LIN {X 0,Y 474.681,Z 256.169,A -85,B 0,C 180,E1 -7215.456,E2 -7215.456} C_VEL
LIN {X 0,Y 474.597,Z 256.179,A -85,B 0,C 180,E1 -7219.013,E2 -7219.013} C_VEL
LIN {X 0,Y 474.568,Z 256.186,A -85,B 0,C 180,E1 -7221.73,E2 -7221.73} C_VEL
LIN {X 0,Y 474.615,Z 256.175,A -85,B 0,C 180,E1 -7224.495,E2 -7224.495} C_VEL
LIN {X 0,Y 474.59,Z 256.182,A -85,B 0,C 180,E1 -7227.327,E2 -7227.327} C_VEL
LIN {X 0,Y 474.543,Z 256.184,A -85,B 0,C 180,E1 -7230.234,E2 -7230.234} C_VEL
LIN {X 0,Y 474.608,Z 256.18,A -85,B 0,C 180,E1 -7233.223,E2 -7233.223} C_VEL
LIN {X 0,Y 474.566,Z 256.181,A -85,B 0,C 180,E1 -7236.325,E2 -7236.325} C_VEL
LIN {X 0,Y 474.594,Z 256.179,A -85,B 0,C 180,E1 -7239.644,E2 -7239.644} C_VEL
LIN {X 0,Y 474.564,Z 256.185,A -85,B 0,C 180,E1 -7242.94,E2 -7242.94} C_VEL
LIN {X 0,Y 474.575,Z 256.179,A -85,B 0,C 180,E1 -7245.892,E2 -7245.892} C_VEL
LIN {X 0,Y 474.594,Z 256.183,A -85,B 0,C 180,E1 -7249.045,E2 -7249.045} C_VEL
LIN {X 0,Y 474.585,Z 256.178,A -85,B 0,C 180,E1 -7251.708,E2 -7251.708} C_VEL
LIN {X 0,Y 474.604,Z 256.181,A -85,B 0,C 180,E1 -7254.725,E2 -7254.725} C_VEL
LIN {X 0,Y 474.605,Z 256.175,A -85,B 0,C 180,E1 -7257.786,E2 -7257.786} C_VEL
LIN {X 0,Y 474.571,Z 256.185,A -85,B 0,C 180,E1 -7260.896,E2 -7260.896} C_VEL
LIN {X 0,Y 474.567,Z 256.182,A -85,B 0,C 180,E1 -7263.623,E2 -7263.623} C_VEL
LIN {X 0,Y 474.649,Z 256.338,A -85,B 0,C 180,E1 -7265.391,E2 -7265.391} C_VEL
LIN {X 0,Y 475.967,Z 264.349,A -85,B 0,C 180,E1 -7266.966,E2 -7266.966} C_VEL
LIN {X 0,Y 475.506,Z 278.927,A -85,B 0,C 180,E1 -7269.676,E2 -7269.676} C_VEL
LIN {X 0,Y 475.135,Z 292.245,A -85,B 0,C 180,E1 -7272.127,E2 -7272.127} C_VEL
LIN {X 0,Y 474.672,Z 310.333,A -85,B 0,C 180,E1 -7275.422,E2 -7275.422} C_VEL
LIN {X 0,Y 474.437,Z 318.145,A -85,B 0,C 180,E1 -7276.819,E2 -7276.819} C_VEL
LIN {X 0,Y 476.321,Z 335.84,A -85,B 0,C 180,E1 -7277.139,E2 -7277.139} C_VEL
LIN {X 0,Y 475.981,Z 395.396,A -85,B 0,C 180,E1 -7278.051,E2 -7278.051} C_VEL
LIN {X 0,Y 475.775,Z 405.125,A -85,B 0,C 180,E1 -7278.309,E2 -7278.309} C_VEL
LIN {X 0,Y 475.51,Z 415.201,A -85,B 0,C 180,E1 -7278.707,E2 -7278.707} C_VEL
LIN {X 0,Y 475.139,Z 426.652,A -85,B 0,C 180,E1 -7279.346,E2 -7279.346} C_VEL
LIN {X 0,Y 474.877,Z 435.271,A -85,B 0,C 180,E1 -7279.986,E2 -7279.986} C_VEL
LIN {X 0,Y 474.58,Z 443.381,A -85,B 0,C 180,E1 -7280.733,E2 -7280.733} C_VEL
LIN {X 0,Y 474.351,Z 450.086,A -85,B 0,C 180,E1 -7281.48,E2 -7281.48} C_VEL
LIN {X 0,Y 474.147,Z 456.454,A -85,B 0,C 180,E1 -7282.334,E2 -7282.334} C_VEL
LIN {X 0,Y 474.037,Z 461.751,A -85,B 0,C 180,E1 -7283.189,E2 -7283.189} C_VEL
LIN {X 0,Y 473.901,Z 466.167,A -85,B 0,C 180,E1 -7284.042,E2 -7284.042} C_VEL
LIN {X 0,Y 473.795,Z 471.377,A -85,B 0,C 180,E1 -7285.321,E2 -7285.321} C_VEL
LIN {X 0,Y 473.848,Z 475.21,A -85,B 0,C 180,E1 -7286.599,E2 -7286.599} C_VEL
LIN {X 0,Y 473.786,Z 476.969,A -85,B 0,C 180,E1 -7287.45,E2 -7287.45} C_VEL
LIN {X 0,Y 473.757,Z 478.23,A -85,B 0,C 180,E1 -7288.3,E2 -7288.3} C_VEL
LIN {X 0,Y 473.695,Z 479.012,A -85,B 0,C 180,E1 -7289.15,E2 -7289.15} C_VEL
LIN {X 0,Y 473.684,Z 479.309,A -85,B 0,C 180,E1 -7290,E2 -7290} C_VEL
LIN {X 0,Y 473.695,Z 479.011,A -85,B 0,C 180,E1 -7290.851,E2 -7290.851} C_VEL
LIN {X 0,Y 473.757,Z 478.227,A -85,B 0,C 180,E1 -7291.701,E2 -7291.701} C_VEL
LIN {X 0,Y 473.787,Z 476.965,A -85,B 0,C 180,E1 -7292.551,E2 -7292.551} C_VEL
LIN {X 0,Y 473.842,Z 474.041,A -85,B 0,C 180,E1 -7293.827,E2 -7293.827} C_VEL
LIN {X 0,Y 473.795,Z 471.371,A -85,B 0,C 180,E1 -7294.68,E2 -7294.68} C_VEL
LIN {X 0,Y 473.9,Z 466.157,A -85,B 0,C 180,E1 -7295.959,E2 -7295.959} C_VEL
LIN {X 0,Y 474.108,Z 459.292,A -85,B 0,C 180,E1 -7297.239,E2 -7297.239} C_VEL
LIN {X 0,Y 474.301,Z 451.789,A -85,B 0,C 180,E1 -7298.307,E2 -7298.307} C_VEL
LIN {X 0,Y 474.532,Z 444.396,A -85,B 0,C 180,E1 -7299.162,E2 -7299.162} C_VEL
LIN {X 0,Y 474.818,Z 436.486,A -85,B 0,C 180,E1 -7299.908,E2 -7299.908} C_VEL
LIN {X 0,Y 475.064,Z 428.131,A -85,B 0,C 180,E1 -7300.549,E2 -7300.549} C_VEL
LIN {X 0,Y 475.485,Z 417.478,A -85,B 0,C 180,E1 -7301.187,E2 -7301.187} C_VEL
LIN {X 0,Y 475.719,Z 406.729,A -85,B 0,C 180,E1 -7301.64,E2 -7301.64} C_VEL
LIN {X 0,Y 475.995,Z 396.227,A -85,B 0,C 180,E1 -7301.93,E2 -7301.93} C_VEL
LIN {X 0,Y 476.23,Z 334.22,A -85,B 0,C 180,E1 -7302.887,E2 -7302.887} C_VEL
LIN {X 0,Y 474.453,Z 318.027,A -85,B 0,C 180,E1 -7303.184,E2 -7303.184} C_VEL
LIN {X 0,Y 474.813,Z 302.683,A -85,B 0,C 180,E1 -7305.967,E2 -7305.967} C_VEL
LIN {X 0,Y 475.369,Z 286.185,A -85,B 0,C 180,E1 -7308.981,E2 -7308.981} C_VEL
LIN {X 0,Y 475.865,Z 269.199,A -85,B 0,C 180,E1 -7312.124,E2 -7312.124} C_VEL
LIN {X 0,Y 475.822,Z 263.099,A -85,B 0,C 180,E1 -7313.273,E2 -7313.273} C_VEL
LIN {X 0,Y 474.632,Z 256.175,A -85,B 0,C 180,E1 -7314.67,E2 -7314.67} C_VEL
LIN {X 0,Y 474.588,Z 256.177,A -85,B 0,C 180,E1 -7318.287,E2 -7318.287} C_VEL
LIN {X 0,Y 474.573,Z 256.186,A -85,B 0,C 180,E1 -7321.22,E2 -7321.22} C_VEL
LIN {X 0,Y 474.604,Z 256.175,A -85,B 0,C 180,E1 -7324.244,E2 -7324.244} C_VEL
LIN {X 0,Y 474.533,Z 256.188,A -85,B 0,C 180,E1 -7327.389,E2 -7327.389} C_VEL
LIN {X 0,Y 474.578,Z 256.18,A -85,B 0,C 180,E1 -7329.64,E2 -7329.64} C_VEL
LIN {X 0,Y 474.565,Z 256.187,A -85,B 0,C 180,E1 -7332.94,E2 -7332.94} C_VEL
LIN {X 0,Y 474.58,Z 256.179,A -85,B 0,C 180,E1 -7335.892,E2 -7335.892} C_VEL
LIN {X 0,Y 474.586,Z 256.182,A -85,B 0,C 180,E1 -7339.047,E2 -7339.047} C_VEL
LIN {X 0,Y 474.586,Z 256.178,A -85,B 0,C 180,E1 -7341.708,E2 -7341.708} C_VEL
LIN {X 0,Y 474.607,Z 256.182,A -85,B 0,C 180,E1 -7344.724,E2 -7344.724} C_VEL
LIN {X 0,Y 474.609,Z 256.175,A -85,B 0,C 180,E1 -7347.786,E2 -7347.786} C_VEL
LIN {X 0,Y 474.575,Z 256.183,A -85,B 0,C 180,E1 -7350.896,E2 -7350.896} C_VEL
LIN {X 0,Y 474.571,Z 256.18,A -85,B 0,C 180,E1 -7353.623,E2 -7353.623} C_VEL
LIN {X 0,Y 474.596,Z 256.181,A -85,B 0,C 180,E1 -7356.653,E2 -7356.653} C_VEL
LIN {X 0,Y 474.586,Z 256.181,A -85,B 0,C 180,E1 -7360.087,E2 -7360.087} C_VEL
LIN {X 0,Y 474.582,Z 256.181,A -85,B 0,C 180,E1 -7362.772,E2 -7362.772} C_VEL
LIN {X 0,Y 474.601,Z 256.177,A -85,B 0,C 180,E1 -7365.42,E2 -7365.42} C_VEL
LIN {X 0,Y 474.685,Z 256.171,A -85,B 0,C 180,E1 -7368.037,E2 -7368.037} C_VEL
LIN {X 0,Y 474.661,Z 256.17,A -85,B 0,C 180,E1 -7371.485,E2 -7371.485} C_VEL
LIN {X 0,Y 474.735,Z 256.165,A -85,B 0,C 180,E1 -7374.052,E2 -7374.052} C_VEL
LIN {X 0,Y 474.871,Z 256.144,A -85,B 0,C 180,E1 -7377.455,E2 -7377.455} C_VEL
LIN {X 0,Y 474.88,Z 256.146,A -85,B 0,C 180,E1 -7380,E2 -7380} C_VEL
LIN {X 0,Y 474.871,Z 256.146,A -85,B 0,C 180,E1 -7382.545,E2 -7382.545} C_VEL
LIN {X 0,Y 474.736,Z 256.163,A -85,B 0,C 180,E1 -7385.948,E2 -7385.948} C_VEL
LIN {X 0,Y 474.662,Z 256.172,A -85,B 0,C 180,E1 -7388.515,E2 -7388.515} C_VEL
LIN {X 0,Y 474.694,Z 256.168,A -85,B 0,C 180,E1 -7391.963,E2 -7391.963} C_VEL
LIN {X 0,Y 474.689,Z 256.17,A -85,B 0,C 180,E1 -7395.456,E2 -7395.456} C_VEL
LIN {X 0,Y 474.604,Z 256.178,A -85,B 0,C 180,E1 -7399.013,E2 -7399.013} C_VEL
LIN {X 0,Y 474.576,Z 256.183,A -85,B 0,C 180,E1 -7401.73,E2 -7401.73} C_VEL
LIN {X 0,Y 474.626,Z 256.175,A -85,B 0,C 180,E1 -7404.495,E2 -7404.495} C_VEL
LIN {X 0,Y 474.598,Z 256.181,A -85,B 0,C 180,E1 -7407.326,E2 -7407.326} C_VEL
LIN {X 0,Y 474.585,Z 256.18,A -85,B 0,C 180,E1 -7410.232,E2 -7410.232} C_VEL
LIN {X 0,Y 474.616,Z 256.178,A -85,B 0,C 180,E1 -7413.222,E2 -7413.222} C_VEL
LIN {X 0,Y 474.583,Z 256.18,A -85,B 0,C 180,E1 -7416.324,E2 -7416.324} C_VEL
LIN {X 0,Y 474.602,Z 256.181,A -85,B 0,C 180,E1 -7419.643,E2 -7419.643} C_VEL
LIN {X 0,Y 474.57,Z 256.184,A -85,B 0,C 180,E1 -7422.939,E2 -7422.939} C_VEL
LIN {X 0,Y 474.603,Z 256.178,A -85,B 0,C 180,E1 -7425.894,E2 -7425.894} C_VEL
LIN {X 0,Y 474.592,Z 256.182,A -85,B 0,C 180,E1 -7429.339,E2 -7429.339} C_VEL
LIN {X 0,Y 474.607,Z 256.178,A -85,B 0,C 180,E1 -7431.705,E2 -7431.705} C_VEL
LIN {X 0,Y 474.621,Z 256.177,A -85,B 0,C 180,E1 -7434.725,E2 -7434.725} C_VEL
LIN {X 0,Y 474.623,Z 256.175,A -85,B 0,C 180,E1 -7437.786,E2 -7437.786} C_VEL
LIN {X 0,Y 474.595,Z 256.181,A -85,B 0,C 180,E1 -7440.891,E2 -7440.891} C_VEL
LIN {X 0,Y 474.591,Z 256.179,A -85,B 0,C 180,E1 -7443.624,E2 -7443.624} C_VEL
LIN {X 0,Y 474.635,Z 256.175,A -85,B 0,C 180,E1 -7446.642,E2 -7446.642} C_VEL
LIN {X 0,Y 474.65,Z 256.173,A -85,B 0,C 180,E1 -7450.089,E2 -7450.089} C_VEL
LIN {X 0,Y 474.642,Z 256.172,A -85,B 0,C 180,E1 -7451.629,E2 -7451.629} C_VEL
LIN {X 0,Y 473.94,Z 256.262,A -85,B 0,C 180,E1 -7452.101,E2 -7452.101} C_VEL
LIN {X 0,Y 471.046,Z 256.625,A -85,B 0,C 180,E1 -7452.839,E2 -7452.839} C_VEL
LIN {X 0,Y 468.163,Z 256.982,A -85,B 0,C 180,E1 -7453.585,E2 -7453.585} C_VEL
LIN {X 0,Y 467.499,Z 257.066,A -85,B 0,C 180,E1 -7454.067,E2 -7454.067} C_VEL
LIN {X 0,Y 467.577,Z 257.787,A -85,B 0,C 180,E1 -7454.302,E2 -7454.302} C_VEL
LIN {X 0,Y 467.519,Z 268.24,A -85,B 0,C 180,E1 -7456.658,E2 -7456.658} C_VEL
LIN {X 0,Y 469.716,Z 281.044,A -85,B 0,C 180,E1 -7456.941,E2 -7456.941} C_VEL
LIN {X 0,Y 469.21,Z 344.335,A -85,B 0,C 180,E1 -7457.922,E2 -7457.922} C_VEL
LIN {X 0,Y 469.077,Z 353.451,A -85,B 0,C 180,E1 -7458.166,E2 -7458.166} C_VEL
LIN {X 0,Y 468.936,Z 363.039,A -85,B 0,C 180,E1 -7458.546,E2 -7458.546} C_VEL
LIN {X 0,Y 468.714,Z 373.066,A -85,B 0,C 180,E1 -7459.088,E2 -7459.088} C_VEL
LIN {X 0,Y 468.48,Z 383.462,A -85,B 0,C 180,E1 -7459.847,E2 -7459.847} C_VEL
LIN {X 0,Y 468.128,Z 391.587,A -85,B 0,C 180,E1 -7460.603,E2 -7460.603} C_VEL
LIN {X 0,Y 467.835,Z 398.286,A -85,B 0,C 180,E1 -7461.36,E2 -7461.36} C_VEL
LIN {X 0,Y 467.558,Z 404.624,A -85,B 0,C 180,E1 -7462.225,E2 -7462.225} C_VEL
LIN {X 0,Y 467.426,Z 409.885,A -85,B 0,C 180,E1 -7463.091,E2 -7463.091} C_VEL
LIN {X 0,Y 467.161,Z 414.285,A -85,B 0,C 180,E1 -7463.955,E2 -7463.955} C_VEL
LIN {X 0,Y 467.088,Z 419.44,A -85,B 0,C 180,E1 -7465.253,E2 -7465.253} C_VEL
LIN {X 0,Y 466.948,Z 422.096,A -85,B 0,C 180,E1 -7466.116,E2 -7466.116} C_VEL
LIN {X 0,Y 466.845,Z 424.999,A -85,B 0,C 180,E1 -7467.411,E2 -7467.411} C_VEL
LIN {X 0,Y 466.704,Z 426.276,A -85,B 0,C 180,E1 -7468.274,E2 -7468.274} C_VEL
LIN {X 0,Y 466.636,Z 427.083,A -85,B 0,C 180,E1 -7469.137,E2 -7469.137} C_VEL
LIN {X 0,Y 466.621,Z 427.39,A -85,B 0,C 180,E1 -7470,E2 -7470} C_VEL
LIN {X 0,Y 466.636,Z 427.117,A -85,B 0,C 180,E1 -7470.863,E2 -7470.863} C_VEL
LIN {X 0,Y 466.705,Z 426.378,A -85,B 0,C 180,E1 -7471.725,E2 -7471.725} C_VEL
LIN {X 0,Y 466.844,Z 425.171,A -85,B 0,C 180,E1 -7472.588,E2 -7472.588} C_VEL
LIN {X 0,Y 466.945,Z 422.341,A -85,B 0,C 180,E1 -7473.883,E2 -7473.883} C_VEL
LIN {X 0,Y 467.069,Z 419.763,A -85,B 0,C 180,E1 -7474.747,E2 -7474.747} C_VEL
LIN {X 0,Y 467.154,Z 414.693,A -85,B 0,C 180,E1 -7476.045,E2 -7476.045} C_VEL
LIN {X 0,Y 467.456,Z 409.234,A -85,B 0,C 180,E1 -7477.123,E2 -7477.123} C_VEL
LIN {X 0,Y 467.696,Z 402.363,A -85,B 0,C 180,E1 -7478.207,E2 -7478.207} C_VEL
LIN {X 0,Y 467.994,Z 394.477,A -85,B 0,C 180,E1 -7479.181,E2 -7479.181} C_VEL
LIN {X 0,Y 468.331,Z 386.948,A -85,B 0,C 180,E1 -7479.937,E2 -7479.937} C_VEL
LIN {X 0,Y 468.521,Z 379.064,A -85,B 0,C 180,E1 -7480.588,E2 -7480.588} C_VEL
LIN {X 0,Y 468.804,Z 370.915,A -85,B 0,C 180,E1 -7481.128,E2 -7481.128} C_VEL
LIN {X 0,Y 469.019,Z 362.665,A -85,B 0,C 180,E1 -7481.561,E2 -7481.561} C_VEL
LIN {X 0,Y 469.096,Z 353.77,A -85,B 0,C 180,E1 -7481.915,E2 -7481.915} C_VEL
LIN {X 0,Y 469.262,Z 344.657,A -85,B 0,C 180,E1 -7482.161,E2 -7482.161} C_VEL
LIN {X 0,Y 469.554,Z 279.505,A -85,B 0,C 180,E1 -7483.179,E2 -7483.179} C_VEL
LIN {X 0,Y 467.522,Z 268.288,A -85,B 0,C 180,E1 -7483.427,E2 -7483.427} C_VEL
LIN {X 0,Y 467.464,Z 257.074,A -85,B 0,C 180,E1 -7485.977,E2 -7485.977} C_VEL
LIN {X 0,Y 467.608,Z 257.049,A -85,B 0,C 180,E1 -7488.761,E2 -7488.761} C_VEL
LIN {X 0,Y 467.57,Z 257.057,A -85,B 0,C 180,E1 -7491.264,E2 -7491.264} C_VEL
LIN {X 0,Y 467.549,Z 257.057,A -85,B 0,C 180,E1 -7493.944,E2 -7493.944} C_VEL
LIN {X 0,Y 467.533,Z 257.061,A -85,B 0,C 180,E1 -7496.805,E2 -7496.805} C_VEL
LIN {X 0,Y 467.53,Z 257.06,A -85,B 0,C 180,E1 -7499.739,E2 -7499.739} C_VEL
LIN {X 0,Y 467.57,Z 257.057,A -85,B 0,C 180,E1 -7502.759,E2 -7502.759} C_VEL
LIN {X 0,Y 467.546,Z 257.057,A -85,B 0,C 180,E1 -7505.89,E2 -7505.89} C_VEL
LIN {X 0,Y 467.549,Z 257.058,A -85,B 0,C 180,E1 -7509.147,E2 -7509.147} C_VEL
LIN {X 0,Y 467.555,Z 257.058,A -85,B 0,C 180,E1 -7511.404,E2 -7511.404} C_VEL
LIN {X 0,Y 467.561,Z 257.056,A -85,B 0,C 180,E1 -7515.052,E2 -7515.052} C_VEL
LIN {X 0,Y 467.556,Z 257.057,A -85,B 0,C 180,E1 -7518.725,E2 -7518.725} C_VEL
LIN {X 0,Y 467.55,Z 257.057,A -85,B 0,C 180,E1 -7521.954,E2 -7521.954} C_VEL
LIN {X 0,Y 467.55,Z 257.058,A -85,B 0,C 180,E1 -7525.166,E2 -7525.166} C_VEL
LIN {X 0,Y 467.552,Z 257.058,A -85,B 0,C 180,E1 -7528.257,E2 -7528.257} C_VEL
LIN {X 0,Y 467.534,Z 257.059,A -85,B 0,C 180,E1 -7531.247,E2 -7531.247} C_VEL
LIN {X 0,Y 467.572,Z 257.055,A -85,B 0,C 180,E1 -7534.401,E2 -7534.401} C_VEL
LIN {X 0,Y 467.563,Z 257.056,A -85,B 0,C 180,E1 -7536.995,E2 -7536.995} C_VEL
LIN {X 0,Y 467.605,Z 257.051,A -85,B 0,C 180,E1 -7539.776,E2 -7539.776} C_VEL
LIN {X 0,Y 467.562,Z 257.057,A -85,B 0,C 180,E1 -7542.505,E2 -7542.505} C_VEL
LIN {X 0,Y 467.585,Z 257.052,A -85,B 0,C 180,E1 -7545.196,E2 -7545.196} C_VEL
LIN {X 0,Y 467.642,Z 257.046,A -85,B 0,C 180,E1 -7547.854,E2 -7547.854} C_VEL
LIN {X 0,Y 467.627,Z 257.047,A -85,B 0,C 180,E1 -7551.356,E2 -7551.356} C_VEL
LIN {X 0,Y 467.697,Z 257.039,A -85,B 0,C 180,E1 -7553.962,E2 -7553.962} C_VEL
LIN {X 0,Y 467.806,Z 257.026,A -85,B 0,C 180,E1 -7557.417,E2 -7557.417} C_VEL
LIN {X 0,Y 467.843,Z 257.022,A -85,B 0,C 180,E1 -7560,E2 -7560} C_VEL
LIN {X 0,Y 467.806,Z 257.025,A -85,B 0,C 180,E1 -7562.583,E2 -7562.583} C_VEL
LIN {X 0,Y 467.694,Z 257.043,A -85,B 0,C 180,E1 -7566.038,E2 -7566.038} C_VEL
LIN {X 0,Y 467.626,Z 257.046,A -85,B 0,C 180,E1 -7568.644,E2 -7568.644} C_VEL
LIN {X 0,Y 467.642,Z 257.045,A -85,B 0,C 180,E1 -7572.354,E2 -7572.354} C_VEL
LIN {X 0,Y 467.594,Z 257.055,A -85,B 0,C 180,E1 -7575.863,E2 -7575.863} C_VEL
LIN {X 0,Y 467.546,Z 257.058,A -85,B 0,C 180,E1 -7579.311,E2 -7579.311} C_VEL
LIN {X 0,Y 467.514,Z 257.061,A -85,B 0,C 180,E1 -7582.075,E2 -7582.075} C_VEL
LIN {X 0,Y 467.55,Z 257.056,A -85,B 0,C 180,E1 -7584.89,E2 -7584.89} C_VEL
LIN {X 0,Y 467.533,Z 257.06,A -85,B 0,C 180,E1 -7587.775,E2 -7587.775} C_VEL
LIN {X 0,Y 467.523,Z 257.061,A -85,B 0,C 180,E1 -7591.037,E2 -7591.037} C_VEL
LIN {X 0,Y 467.56,Z 257.055,A -85,B 0,C 180,E1 -7593.79,E2 -7593.79} C_VEL
LIN {X 0,Y 467.5,Z 257.064,A -85,B 0,C 180,E1 -7596.965,E2 -7596.965} C_VEL
LIN {X 0,Y 467.555,Z 257.054,A -85,B 0,C 180,E1 -7599.951,E2 -7599.951} C_VEL
LIN {X 0,Y 467.513,Z 257.06,A -85,B 0,C 180,E1 -7602.568,E2 -7602.568} C_VEL
LIN {X 0,Y 467.559,Z 257.06,A -85,B 0,C 180,E1 -7605.053,E2 -7605.053} C_VEL
LIN {X 0,Y 467.555,Z 257.057,A -85,B 0,C 180,E1 -7608.726,E2 -7608.726} C_VEL
LIN {X 0,Y 467.535,Z 257.056,A -85,B 0,C 180,E1 -7611.953,E2 -7611.953} C_VEL
LIN {X 0,Y 467.54,Z 257.058,A -85,B 0,C 180,E1 -7615.166,E2 -7615.166} C_VEL
LIN {X 0,Y 467.538,Z 257.057,A -85,B 0,C 180,E1 -7618.257,E2 -7618.257} C_VEL
LIN {X 0,Y 467.52,Z 257.06,A -85,B 0,C 180,E1 -7621.247,E2 -7621.247} C_VEL
LIN {X 0,Y 467.558,Z 257.059,A -85,B 0,C 180,E1 -7624.406,E2 -7624.406} C_VEL
LIN {X 0,Y 467.598,Z 257.157,A -85,B 0,C 180,E1 -7625.232,E2 -7625.232} C_VEL
LIN {X 0,Y 468.96,Z 265.186,A -85,B 0,C 180,E1 -7626.838,E2 -7626.838} C_VEL
LIN {X 0,Y 468.586,Z 278.538,A -85,B 0,C 180,E1 -7629.363,E2 -7629.363} C_VEL
LIN {X 0,Y 468.1,Z 293.061,A -85,B 0,C 180,E1 -7632.075,E2 -7632.075} C_VEL
LIN {X 0,Y 467.656,Z 309.939,A -85,B 0,C 180,E1 -7635.199,E2 -7635.199} C_VEL
LIN {X 0,Y 467.41,Z 317.763,A -85,B 0,C 180,E1 -7636.617,E2 -7636.617} C_VEL
LIN {X 0,Y 469.384,Z 335.605,A -85,B 0,C 180,E1 -7636.947,E2 -7636.947} C_VEL
LIN {X 0,Y 469.034,Z 395.056,A -85,B 0,C 180,E1 -7637.873,E2 -7637.873} C_VEL
LIN {X 0,Y 468.823,Z 404.74,A -85,B 0,C 180,E1 -7638.133,E2 -7638.133} C_VEL
LIN {X 0,Y 468.544,Z 414.814,A -85,B 0,C 180,E1 -7638.537,E2 -7638.537} C_VEL
LIN {X 0,Y 468.151,Z 426.262,A -85,B 0,C 180,E1 -7639.185,E2 -7639.185} C_VEL
LIN {X 0,Y 467.854,Z 434.879,A -85,B 0,C 180,E1 -7639.834,E2 -7639.834} C_VEL
LIN {X 0,Y 467.553,Z 442.99,A -85,B 0,C 180,E1 -7640.592,E2 -7640.592} C_VEL
LIN {X 0,Y 467.291,Z 449.694,A -85,B 0,C 180,E1 -7641.35,E2 -7641.35} C_VEL
LIN {X 0,Y 467.076,Z 456.061,A -85,B 0,C 180,E1 -7642.218,E2 -7642.218} C_VEL
LIN {X 0,Y 466.991,Z 461.36,A -85,B 0,C 180,E1 -7643.086,E2 -7643.086} C_VEL
LIN {X 0,Y 466.811,Z 465.774,A -85,B 0,C 180,E1 -7643.951,E2 -7643.951} C_VEL
LIN {X 0,Y 466.721,Z 470.986,A -85,B 0,C 180,E1 -7645.25,E2 -7645.25} C_VEL
LIN {X 0,Y 466.761,Z 474.818,A -85,B 0,C 180,E1 -7646.548,E2 -7646.548} C_VEL
LIN {X 0,Y 466.705,Z 476.578,A -85,B 0,C 180,E1 -7647.411,E2 -7647.411} C_VEL
LIN {X 0,Y 466.692,Z 477.84,A -85,B 0,C 180,E1 -7648.275,E2 -7648.275} C_VEL
LIN {X 0,Y 466.625,Z 478.622,A -85,B 0,C 180,E1 -7649.137,E2 -7649.137} C_VEL
LIN {X 0,Y 466.612,Z 478.918,A -85,B 0,C 180,E1 -7650,E2 -7650} C_VEL
LIN {X 0,Y 466.625,Z 478.621,A -85,B 0,C 180,E1 -7650.863,E2 -7650.863} C_VEL
LIN {X 0,Y 466.692,Z 477.837,A -85,B 0,C 180,E1 -7651.726,E2 -7651.726} C_VEL
LIN {X 0,Y 466.705,Z 476.573,A -85,B 0,C 180,E1 -7652.59,E2 -7652.59} C_VEL
LIN {X 0,Y 466.732,Z 473.647,A -85,B 0,C 180,E1 -7653.886,E2 -7653.886} C_VEL
LIN {X 0,Y 466.721,Z 470.978,A -85,B 0,C 180,E1 -7654.751,E2 -7654.751} C_VEL
LIN {X 0,Y 466.81,Z 465.762,A -85,B 0,C 180,E1 -7656.05,E2 -7656.05} C_VEL
LIN {X 0,Y 467.041,Z 458.897,A -85,B 0,C 180,E1 -7657.349,E2 -7657.349} C_VEL
LIN {X 0,Y 467.237,Z 451.394,A -85,B 0,C 180,E1 -7658.434,E2 -7658.434} C_VEL
LIN {X 0,Y 467.505,Z 444.001,A -85,B 0,C 180,E1 -7659.3,E2 -7659.3} C_VEL
LIN {X 0,Y 467.825,Z 436.092,A -85,B 0,C 180,E1 -7660.058,E2 -7660.058} C_VEL
LIN {X 0,Y 468.085,Z 427.736,A -85,B 0,C 180,E1 -7660.708,E2 -7660.708} C_VEL
LIN {X 0,Y 468.52,Z 417.081,A -85,B 0,C 180,E1 -7661.355,E2 -7661.355} C_VEL
LIN {X 0,Y 468.77,Z 406.33,A -85,B 0,C 180,E1 -7661.815,E2 -7661.815} C_VEL
LIN {X 0,Y 469.054,Z 395.824,A -85,B 0,C 180,E1 -7662.109,E2 -7662.109} C_VEL
LIN {X 0,Y 469.386,Z 335.429,A -85,B 0,C 180,E1 -7663.054,E2 -7663.054} C_VEL
LIN {X 0,Y 467.395,Z 317.627,A -85,B 0,C 180,E1 -7663.386,E2 -7663.386} C_VEL
LIN {X 0,Y 467.72,Z 303.904,A -85,B 0,C 180,E1 -7665.915,E2 -7665.915} C_VEL
LIN {X 0,Y 468.338,Z 287.148,A -85,B 0,C 180,E1 -7669.022,E2 -7669.022} C_VEL
LIN {X 0,Y 468.895,Z 270.019,A -85,B 0,C 180,E1 -7672.239,E2 -7672.239} C_VEL
LIN {X 0,Y 468.82,Z 263.978,A -85,B 0,C 180,E1 -7673.396,E2 -7673.396} C_VEL
LIN {X 0,Y 467.584,Z 257.054,A -85,B 0,C 180,E1 -7674.829,E2 -7674.829} C_VEL
LIN {X 0,Y 467.537,Z 257.059,A -85,B 0,C 180,E1 -7677.775,E2 -7677.775} C_VEL
LIN {X 0,Y 467.527,Z 257.061,A -85,B 0,C 180,E1 -7681.037,E2 -7681.037} C_VEL
LIN {X 0,Y 467.562,Z 257.052,A -85,B 0,C 180,E1 -7684.238,E2 -7684.238} C_VEL
LIN {X 0,Y 467.51,Z 257.066,A -85,B 0,C 180,E1 -7687.18,E2 -7687.18} C_VEL
LIN {X 0,Y 467.517,Z 257.058,A -85,B 0,C 180,E1 -7690.271,E2 -7690.271} C_VEL
LIN {X 0,Y 467.516,Z 257.06,A -85,B 0,C 180,E1 -7692.569,E2 -7692.569} C_VEL
LIN {X 0,Y 467.562,Z 257.058,A -85,B 0,C 180,E1 -7695.052,E2 -7695.052} C_VEL
LIN {X 0,Y 467.554,Z 257.059,A -85,B 0,C 180,E1 -7698.727,E2 -7698.727} C_VEL
LIN {X 0,Y 467.537,Z 257.056,A -85,B 0,C 180,E1 -7701.953,E2 -7701.953} C_VEL
LIN {X 0,Y 467.543,Z 257.057,A -85,B 0,C 180,E1 -7705.166,E2 -7705.166} C_VEL
LIN {X 0,Y 467.542,Z 257.058,A -85,B 0,C 180,E1 -7708.257,E2 -7708.257} C_VEL
LIN {X 0,Y 467.524,Z 257.059,A -85,B 0,C 180,E1 -7711.247,E2 -7711.247} C_VEL
LIN {X 0,Y 467.561,Z 257.059,A -85,B 0,C 180,E1 -7714.406,E2 -7714.406} C_VEL
LIN {X 0,Y 467.546,Z 257.057,A -85,B 0,C 180,E1 -7716.994,E2 -7716.994} C_VEL
LIN {X 0,Y 467.538,Z 257.057,A -85,B 0,C 180,E1 -7719.773,E2 -7719.773} C_VEL
LIN {X 0,Y 467.552,Z 257.058,A -85,B 0,C 180,E1 -7722.505,E2 -7722.505} C_VEL
LIN {X 0,Y 467.558,Z 257.055,A -85,B 0,C 180,E1 -7725.195,E2 -7725.195} C_VEL
LIN {X 0,Y 467.642,Z 257.046,A -85,B 0,C 180,E1 -7727.854,E2 -7727.854} C_VEL
LIN {X 0,Y 467.63,Z 257.046,A -85,B 0,C 180,E1 -7731.356,E2 -7731.356} C_VEL
LIN {X 0,Y 467.701,Z 257.041,A -85,B 0,C 180,E1 -7733.962,E2 -7733.962} C_VEL
LIN {X 0,Y 467.812,Z 257.024,A -85,B 0,C 180,E1 -7737.417,E2 -7737.417} C_VEL
LIN {X 0,Y 467.849,Z 257.022,A -85,B 0,C 180,E1 -7740,E2 -7740} C_VEL
LIN {X 0,Y 467.812,Z 257.025,A -85,B 0,C 180,E1 -7742.583,E2 -7742.583} C_VEL
LIN {X 0,Y 467.701,Z 257.039,A -85,B 0,C 180,E1 -7746.038,E2 -7746.038} C_VEL
LIN {X 0,Y 467.631,Z 257.047,A -85,B 0,C 180,E1 -7748.644,E2 -7748.644} C_VEL
LIN {X 0,Y 467.649,Z 257.045,A -85,B 0,C 180,E1 -7752.146,E2 -7752.146} C_VEL
LIN {X 0,Y 467.614,Z 257.05,A -85,B 0,C 180,E1 -7755.696,E2 -7755.696} C_VEL
LIN {X 0,Y 467.573,Z 257.053,A -85,B 0,C 180,E1 -7758.748,E2 -7758.748} C_VEL
LIN {X 0,Y 467.559,Z 257.058,A -85,B 0,C 180,E1 -7761.261,E2 -7761.261} C_VEL
LIN {X 0,Y 467.552,Z 257.058,A -85,B 0,C 180,E1 -7763.945,E2 -7763.945} C_VEL
LIN {X 0,Y 467.536,Z 257.059,A -85,B 0,C 180,E1 -7766.805,E2 -7766.805} C_VEL
LIN {X 0,Y 467.535,Z 257.06,A -85,B 0,C 180,E1 -7769.74,E2 -7769.74} C_VEL
LIN {X 0,Y 467.575,Z 257.054,A -85,B 0,C 180,E1 -7772.759,E2 -7772.759} C_VEL
LIN {X 0,Y 467.55,Z 257.058,A -85,B 0,C 180,E1 -7775.89,E2 -7775.89} C_VEL
LIN {X 0,Y 467.549,Z 257.058,A -85,B 0,C 180,E1 -7779.148,E2 -7779.148} C_VEL
LIN {X 0,Y 467.559,Z 257.057,A -85,B 0,C 180,E1 -7781.405,E2 -7781.405} C_VEL
LIN {X 0,Y 467.566,Z 257.056,A -85,B 0,C 180,E1 -7785.052,E2 -7785.052} C_VEL
LIN {X 0,Y 467.561,Z 257.057,A -85,B 0,C 180,E1 -7788.726,E2 -7788.726} C_VEL
LIN {X 0,Y 467.562,Z 257.055,A -85,B 0,C 180,E1 -7791.955,E2 -7791.955} C_VEL
LIN {X 0,Y 467.557,Z 257.058,A -85,B 0,C 180,E1 -7795.166,E2 -7795.166} C_VEL
LIN {X 0,Y 467.553,Z 257.057,A -85,B 0,C 180,E1 -7798.257,E2 -7798.257} C_VEL
LIN {X 0,Y 467.542,Z 257.06,A -85,B 0,C 180,E1 -7801.248,E2 -7801.248} C_VEL
LIN {X 0,Y 467.579,Z 257.054,A -85,B 0,C 180,E1 -7804.401,E2 -7804.401} C_VEL
LIN {X 0,Y 467.571,Z 257.057,A -85,B 0,C 180,E1 -7806.995,E2 -7806.995} C_VEL
LIN {X 0,Y 467.62,Z 257.047,A -85,B 0,C 180,E1 -7809.777,E2 -7809.777} C_VEL
LIN {X 0,Y 467.566,Z 257.059,A -85,B 0,C 180,E1 -7812.505,E2 -7812.505} C_VEL
LIN {X 0,Y 467.499,Z 257.066,A -85,B 0,C 180,E1 -7814.067,E2 -7814.067} C_VEL
LIN {X 0,Y 467.2,Z 258.222,A -85,B 0,C 180,E1 -7814.386,E2 -7814.386} C_VEL
LIN {X 0,Y 465.318,Z 260.917,A -85,B 0,C 180,E1 -7814.922,E2 -7814.922} C_VEL
LIN {X 0,Y 461.257,Z 265.566,A -85,B 0,C 180,E1 -7815.78,E2 -7815.78} C_VEL
LIN {X 0,Y 460.529,Z 267.456,A -85,B 0,C 180,E1 -7816.195,E2 -7816.195} C_VEL
LIN {X 0,Y 460.511,Z 268.648,A -85,B 0,C 180,E1 -7816.461,E2 -7816.461} C_VEL
LIN {X 0,Y 462.832,Z 281.468,A -85,B 0,C 180,E1 -7816.744,E2 -7816.744} C_VEL
LIN {X 0,Y 462.292,Z 344.747,A -85,B 0,C 180,E1 -7817.739,E2 -7817.739} C_VEL
LIN {X 0,Y 462.15,Z 353.855,A -85,B 0,C 180,E1 -7817.986,E2 -7817.986} C_VEL
LIN {X 0,Y 462.013,Z 363.439,A -85,B 0,C 180,E1 -7818.372,E2 -7818.372} C_VEL
LIN {X 0,Y 461.775,Z 373.464,A -85,B 0,C 180,E1 -7818.922,E2 -7818.922} C_VEL
LIN {X 0,Y 461.505,Z 383.858,A -85,B 0,C 180,E1 -7819.692,E2 -7819.692} C_VEL
LIN {X 0,Y 461.15,Z 391.982,A -85,B 0,C 180,E1 -7820.46,E2 -7820.46} C_VEL
LIN {X 0,Y 460.848,Z 398.68,A -85,B 0,C 180,E1 -7821.228,E2 -7821.228} C_VEL
LIN {X 0,Y 460.549,Z 405.018,A -85,B 0,C 180,E1 -7822.106,E2 -7822.106} C_VEL
LIN {X 0,Y 460.396,Z 410.278,A -85,B 0,C 180,E1 -7822.985,E2 -7822.985} C_VEL
LIN {X 0,Y 460.135,Z 414.677,A -85,B 0,C 180,E1 -7823.862,E2 -7823.862} C_VEL
LIN {X 0,Y 460.041,Z 419.832,A -85,B 0,C 180,E1 -7825.18,E2 -7825.18} C_VEL
LIN {X 0,Y 459.886,Z 422.488,A -85,B 0,C 180,E1 -7826.056,E2 -7826.056} C_VEL
LIN {X 0,Y 459.774,Z 425.39,A -85,B 0,C 180,E1 -7827.371,E2 -7827.371} C_VEL
LIN {X 0,Y 459.644,Z 426.666,A -85,B 0,C 180,E1 -7828.247,E2 -7828.247} C_VEL
LIN {X 0,Y 459.568,Z 427.473,A -85,B 0,C 180,E1 -7829.123,E2 -7829.123} C_VEL
LIN {X 0,Y 459.551,Z 427.78,A -85,B 0,C 180,E1 -7830,E2 -7830} C_VEL
LIN {X 0,Y 459.569,Z 427.507,A -85,B 0,C 180,E1 -7830.876,E2 -7830.876} C_VEL
LIN {X 0,Y 459.644,Z 426.768,A -85,B 0,C 180,E1 -7831.752,E2 -7831.752} C_VEL
LIN {X 0,Y 459.76,Z 425.562,A -85,B 0,C 180,E1 -7832.628,E2 -7832.628} C_VEL
LIN {X 0,Y 459.882,Z 422.73,A -85,B 0,C 180,E1 -7833.943,E2 -7833.943} C_VEL
LIN {X 0,Y 460.016,Z 420.153,A -85,B 0,C 180,E1 -7834.82,E2 -7834.82} C_VEL
LIN {X 0,Y 460.126,Z 415.081,A -85,B 0,C 180,E1 -7836.137,E2 -7836.137} C_VEL
LIN {X 0,Y 460.409,Z 410.018,A -85,B 0,C 180,E1 -7837.158,E2 -7837.158} C_VEL
LIN {X 0,Y 460.674,Z 402.752,A -85,B 0,C 180,E1 -7838.333,E2 -7838.333} C_VEL
LIN {X 0,Y 461.007,Z 394.863,A -85,B 0,C 180,E1 -7839.321,E2 -7839.321} C_VEL
LIN {X 0,Y 461.363,Z 387.334,A -85,B 0,C 180,E1 -7840.089,E2 -7840.089} C_VEL
LIN {X 0,Y 461.578,Z 379.448,A -85,B 0,C 180,E1 -7840.749,E2 -7840.749} C_VEL
LIN {X 0,Y 461.874,Z 371.298,A -85,B 0,C 180,E1 -7841.297,E2 -7841.297} C_VEL
LIN {X 0,Y 462.073,Z 363.047,A -85,B 0,C 180,E1 -7841.737,E2 -7841.737} C_VEL
LIN {X 0,Y 462.17,Z 354.148,A -85,B 0,C 180,E1 -7842.096,E2 -7842.096} C_VEL
LIN {X 0,Y 462.335,Z 345.115,A -85,B 0,C 180,E1 -7842.345,E2 -7842.345} C_VEL
LIN {X 0,Y 462.678,Z 280.292,A -85,B 0,C 180,E1 -7843.372,E2 -7843.372} C_VEL
LIN {X 0,Y 460.505,Z 268.647,A -85,B 0,C 180,E1 -7843.635,E2 -7843.635} C_VEL
LIN {X 0,Y 460.439,Z 257.971,A -85,B 0,C 180,E1 -7846.067,E2 -7846.067} C_VEL
LIN {X 0,Y 460.563,Z 257.928,A -85,B 0,C 180,E1 -7848.898,E2 -7848.898} C_VEL
LIN {X 0,Y 460.512,Z 257.934,A -85,B 0,C 180,E1 -7851.485,E2 -7851.485} C_VEL
LIN {X 0,Y 460.513,Z 257.933,A -85,B 0,C 180,E1 -7854.333,E2 -7854.333} C_VEL
LIN {X 0,Y 460.489,Z 257.938,A -85,B 0,C 180,E1 -7857.249,E2 -7857.249} C_VEL
LIN {X 0,Y 460.491,Z 257.936,A -85,B 0,C 180,E1 -7860.241,E2 -7860.241} C_VEL
LIN {X 0,Y 460.513,Z 257.934,A -85,B 0,C 180,E1 -7863.325,E2 -7863.325} C_VEL
LIN {X 0,Y 460.468,Z 257.94,A -85,B 0,C 180,E1 -7866.529,E2 -7866.529} C_VEL
LIN {X 0,Y 460.509,Z 257.934,A -85,B 0,C 180,E1 -7869.864,E2 -7869.864} C_VEL
LIN {X 0,Y 460.458,Z 257.941,A -85,B 0,C 180,E1 -7872.893,E2 -7872.893} C_VEL
LIN {X 0,Y 460.499,Z 257.935,A -85,B 0,C 180,E1 -7875.831,E2 -7875.831} C_VEL
LIN {X 0,Y 460.51,Z 257.935,A -85,B 0,C 180,E1 -7878.986,E2 -7878.986} C_VEL
LIN {X 0,Y 460.49,Z 257.938,A -85,B 0,C 180,E1 -7882.376,E2 -7882.376} C_VEL
LIN {X 0,Y 460.53,Z 257.931,A -85,B 0,C 180,E1 -7885.622,E2 -7885.622} C_VEL
LIN {X 0,Y 460.499,Z 257.936,A -85,B 0,C 180,E1 -7888.742,E2 -7888.742} C_VEL
LIN {X 0,Y 460.499,Z 257.935,A -85,B 0,C 180,E1 -7891.763,E2 -7891.763} C_VEL
LIN {X 0,Y 460.517,Z 257.935,A -85,B 0,C 180,E1 -7894.703,E2 -7894.703} C_VEL
LIN {X 0,Y 460.497,Z 257.935,A -85,B 0,C 180,E1 -7897.571,E2 -7897.571} C_VEL
LIN {X 0,Y 460.556,Z 257.929,A -85,B 0,C 180,E1 -7900.384,E2 -7900.384} C_VEL
LIN {X 0,Y 460.561,Z 257.928,A -85,B 0,C 180,E1 -7904.057,E2 -7904.057} C_VEL
LIN {X 0,Y 460.597,Z 257.924,A -85,B 0,C 180,E1 -7907.665,E2 -7907.665} C_VEL
LIN {X 0,Y 460.582,Z 257.924,A -85,B 0,C 180,E1 -7911.223,E2 -7911.223} C_VEL
LIN {X 0,Y 460.663,Z 257.915,A -85,B 0,C 180,E1 -7913.869,E2 -7913.869} C_VEL
LIN {X 0,Y 460.749,Z 257.905,A -85,B 0,C 180,E1 -7917.377,E2 -7917.377} C_VEL
LIN {X 0,Y 460.812,Z 257.898,A -85,B 0,C 180,E1 -7920,E2 -7920} C_VEL
LIN {X 0,Y 460.749,Z 257.904,A -85,B 0,C 180,E1 -7922.623,E2 -7922.623} C_VEL
LIN {X 0,Y 460.66,Z 257.918,A -85,B 0,C 180,E1 -7926.13,E2 -7926.13} C_VEL
LIN {X 0,Y 460.581,Z 257.924,A -85,B 0,C 180,E1 -7928.777,E2 -7928.777} C_VEL
LIN {X 0,Y 460.591,Z 257.923,A -85,B 0,C 180,E1 -7932.435,E2 -7932.435} C_VEL
LIN {X 0,Y 460.551,Z 257.931,A -85,B 0,C 180,E1 -7935.978,E2 -7935.978} C_VEL
LIN {X 0,Y 460.524,Z 257.932,A -85,B 0,C 180,E1 -7938.887,E2 -7938.887} C_VEL
LIN {X 0,Y 460.503,Z 257.937,A -85,B 0,C 180,E1 -7941.486,E2 -7941.486} C_VEL
LIN {X 0,Y 460.507,Z 257.933,A -85,B 0,C 180,E1 -7944.334,E2 -7944.334} C_VEL
LIN {X 0,Y 460.483,Z 257.938,A -85,B 0,C 180,E1 -7947.249,E2 -7947.249} C_VEL
LIN {X 0,Y 460.472,Z 257.937,A -85,B 0,C 180,E1 -7950.243,E2 -7950.243} C_VEL
LIN {X 0,Y 460.51,Z 257.937,A -85,B 0,C 180,E1 -7953.326,E2 -7953.326} C_VEL
LIN {X 0,Y 460.454,Z 257.939,A -85,B 0,C 180,E1 -7956.531,E2 -7956.531} C_VEL
LIN {X 0,Y 460.504,Z 257.933,A -85,B 0,C 180,E1 -7959.865,E2 -7959.865} C_VEL
LIN {X 0,Y 460.457,Z 257.942,A -85,B 0,C 180,E1 -7962.894,E2 -7962.894} C_VEL
LIN {X 0,Y 460.499,Z 257.933,A -85,B 0,C 180,E1 -7965.832,E2 -7965.832} C_VEL
LIN {X 0,Y 460.509,Z 257.938,A -85,B 0,C 180,E1 -7968.987,E2 -7968.987} C_VEL
LIN {X 0,Y 460.478,Z 257.937,A -85,B 0,C 180,E1 -7972.375,E2 -7972.375} C_VEL
LIN {X 0,Y 460.52,Z 257.93,A -85,B 0,C 180,E1 -7975.622,E2 -7975.622} C_VEL
LIN {X 0,Y 460.5,Z 257.939,A -85,B 0,C 180,E1 -7978.742,E2 -7978.742} C_VEL
LIN {X 0,Y 460.492,Z 257.935,A -85,B 0,C 180,E1 -7981.764,E2 -7981.764} C_VEL
LIN {X 0,Y 460.546,Z 257.975,A -85,B 0,C 180,E1 -7985.067,E2 -7985.067} C_VEL
LIN {X 0,Y 462.031,Z 267.215,A -85,B 0,C 180,E1 -7986.941,E2 -7986.941} C_VEL
LIN {X 0,Y 461.474,Z 281.781,A -85,B 0,C 180,E1 -7989.729,E2 -7989.729} C_VEL
LIN {X 0,Y 461.017,Z 295.082,A -85,B 0,C 180,E1 -7992.249,E2 -7992.249} C_VEL
LIN {X 0,Y 460.528,Z 311.946,A -85,B 0,C 180,E1 -7995.416,E2 -7995.416} C_VEL
LIN {X 0,Y 460.356,Z 317.38,A -85,B 0,C 180,E1 -7996.408,E2 -7996.408} C_VEL
LIN {X 0,Y 462.495,Z 336.844,A -85,B 0,C 180,E1 -7996.775,E2 -7996.775} C_VEL
LIN {X 0,Y 462.102,Z 394.722,A -85,B 0,C 180,E1 -7997.689,E2 -7997.689} C_VEL
LIN {X 0,Y 461.887,Z 404.356,A -85,B 0,C 180,E1 -7997.952,E2 -7997.952} C_VEL
LIN {X 0,Y 461.565,Z 414.426,A -85,B 0,C 180,E1 -7998.361,E2 -7998.361} C_VEL
LIN {X 0,Y 461.159,Z 425.873,A -85,B 0,C 180,E1 -7999.019,E2 -7999.019} C_VEL
LIN {X 0,Y 460.858,Z 434.49,A -85,B 0,C 180,E1 -7999.678,E2 -7999.678} C_VEL
LIN {X 0,Y 460.542,Z 442.6,A -85,B 0,C 180,E1 -8000.448,E2 -8000.448} C_VEL
LIN {X 0,Y 460.254,Z 449.302,A -85,B 0,C 180,E1 -8001.217,E2 -8001.217} C_VEL
LIN {X 0,Y 460.025,Z 455.67,A -85,B 0,C 180,E1 -8002.097,E2 -8002.097} C_VEL
LIN {X 0,Y 459.936,Z 460.969,A -85,B 0,C 180,E1 -8002.979,E2 -8002.979} C_VEL
LIN {X 0,Y 459.721,Z 465.382,A -85,B 0,C 180,E1 -8003.857,E2 -8003.857} C_VEL
LIN {X 0,Y 459.651,Z 470.595,A -85,B 0,C 180,E1 -8005.177,E2 -8005.177} C_VEL
LIN {X 0,Y 459.659,Z 474.426,A -85,B 0,C 180,E1 -8006.494,E2 -8006.494} C_VEL
LIN {X 0,Y 459.626,Z 476.187,A -85,B 0,C 180,E1 -8007.371,E2 -8007.371} C_VEL
LIN {X 0,Y 459.599,Z 477.448,A -85,B 0,C 180,E1 -8008.248,E2 -8008.248} C_VEL
LIN {X 0,Y 459.558,Z 478.232,A -85,B 0,C 180,E1 -8009.124,E2 -8009.124} C_VEL
LIN {X 0,Y 459.543,Z 478.528,A -85,B 0,C 180,E1 -8010,E2 -8010} C_VEL
LIN {X 0,Y 459.558,Z 478.231,A -85,B 0,C 180,E1 -8010.877,E2 -8010.877} C_VEL
LIN {X 0,Y 459.599,Z 477.445,A -85,B 0,C 180,E1 -8011.753,E2 -8011.753} C_VEL
LIN {X 0,Y 459.627,Z 476.181,A -85,B 0,C 180,E1 -8012.63,E2 -8012.63} C_VEL
LIN {X 0,Y 459.626,Z 473.253,A -85,B 0,C 180,E1 -8013.946,E2 -8013.946} C_VEL
LIN {X 0,Y 459.651,Z 470.586,A -85,B 0,C 180,E1 -8014.824,E2 -8014.824} C_VEL
LIN {X 0,Y 459.719,Z 465.367,A -85,B 0,C 180,E1 -8016.144,E2 -8016.144} C_VEL
LIN {X 0,Y 459.965,Z 458.502,A -85,B 0,C 180,E1 -8017.463,E2 -8017.463} C_VEL
LIN {X 0,Y 460.19,Z 450.998,A -85,B 0,C 180,E1 -8018.564,E2 -8018.564} C_VEL
LIN {X 0,Y 460.487,Z 443.606,A -85,B 0,C 180,E1 -8019.443,E2 -8019.443} C_VEL
LIN {X 0,Y 460.812,Z 435.695,A -85,B 0,C 180,E1 -8020.213,E2 -8020.213} C_VEL
LIN {X 0,Y 461.1,Z 427.34,A -85,B 0,C 180,E1 -8020.873,E2 -8020.873} C_VEL
LIN {X 0,Y 461.553,Z 416.684,A -85,B 0,C 180,E1 -8021.529,E2 -8021.529} C_VEL
LIN {X 0,Y 461.829,Z 405.931,A -85,B 0,C 180,E1 -8021.995,E2 -8021.995} C_VEL
LIN {X 0,Y 462.111,Z 395.419,A -85,B 0,C 180,E1 -8022.294,E2 -8022.294} C_VEL
LIN {X 0,Y 462.478,Z 341.128,A -85,B 0,C 180,E1 -8023.157,E2 -8023.157} C_VEL
LIN {X 0,Y 462.243,Z 334.283,A -85,B 0,C 180,E1 -8023.27,E2 -8023.27} C_VEL
LIN {X 0,Y 460.363,Z 317.23,A -85,B 0,C 180,E1 -8023.595,E2 -8023.595} C_VEL
LIN {X 0,Y 460.818,Z 301.214,A -85,B 0,C 180,E1 -8026.594,E2 -8026.594} C_VEL
LIN {X 0,Y 461.399,Z 285.394,A -85,B 0,C 180,E1 -8029.579,E2 -8029.579} C_VEL
LIN {X 0,Y 461.956,Z 269.623,A -85,B 0,C 180,E1 -8032.591,E2 -8032.591} C_VEL
LIN {X 0,Y 461.948,Z 265.965,A -85,B 0,C 180,E1 -8033.301,E2 -8033.301} C_VEL
LIN {X 0,Y 460.546,Z 257.931,A -85,B 0,C 180,E1 -8034.964,E2 -8034.964} C_VEL
LIN {X 0,Y 460.495,Z 257.933,A -85,B 0,C 180,E1 -8038.237,E2 -8038.237} C_VEL
LIN {X 0,Y 460.495,Z 257.94,A -85,B 0,C 180,E1 -8041.278,E2 -8041.278} C_VEL
LIN {X 0,Y 460.508,Z 257.931,A -85,B 0,C 180,E1 -8044.501,E2 -8044.501} C_VEL
LIN {X 0,Y 460.478,Z 257.937,A -85,B 0,C 180,E1 -8047.626,E2 -8047.626} C_VEL
LIN {X 0,Y 460.499,Z 257.939,A -85,B 0,C 180,E1 -8051.015,E2 -8051.015} C_VEL
LIN {X 0,Y 460.51,Z 257.934,A -85,B 0,C 180,E1 -8054.59,E2 -8054.59} C_VEL
LIN {X 0,Y 460.472,Z 257.936,A -85,B 0,C 180,E1 -8057.813,E2 -8057.813} C_VEL
LIN {X 0,Y 460.495,Z 257.934,A -85,B 0,C 180,E1 -8060.134,E2 -8060.134} C_VEL
LIN {X 0,Y 460.458,Z 257.939,A -85,B 0,C 180,E1 -8063.469,E2 -8063.469} C_VEL
LIN {X 0,Y 460.5,Z 257.939,A -85,B 0,C 180,E1 -8066.673,E2 -8066.673} C_VEL
LIN {X 0,Y 460.478,Z 257.936,A -85,B 0,C 180,E1 -8069.758,E2 -8069.758} C_VEL
LIN {X 0,Y 460.484,Z 257.938,A -85,B 0,C 180,E1 -8072.751,E2 -8072.751} C_VEL
LIN {X 0,Y 460.495,Z 257.934,A -85,B 0,C 180,E1 -8075.665,E2 -8075.665} C_VEL
LIN {X 0,Y 460.51,Z 257.935,A -85,B 0,C 180,E1 -8078.583,E2 -8078.583} C_VEL
LIN {X 0,Y 460.526,Z 257.931,A -85,B 0,C 180,E1 -8081.308,E2 -8081.308} C_VEL
LIN {X 0,Y 460.521,Z 257.934,A -85,B 0,C 180,E1 -8084.056,E2 -8084.056} C_VEL
LIN {X 0,Y 460.602,Z 257.922,A -85,B 0,C 180,E1 -8087.666,E2 -8087.666} C_VEL
LIN {X 0,Y 460.585,Z 257.924,A -85,B 0,C 180,E1 -8091.223,E2 -8091.223} C_VEL
LIN {X 0,Y 460.667,Z 257.917,A -85,B 0,C 180,E1 -8093.87,E2 -8093.87} C_VEL
LIN {X 0,Y 460.755,Z 257.903,A -85,B 0,C 180,E1 -8097.377,E2 -8097.377} C_VEL
LIN {X 0,Y 460.819,Z 257.897,A -85,B 0,C 180,E1 -8100,E2 -8100} C_VEL
LIN {X 0,Y 460.755,Z 257.904,A -85,B 0,C 180,E1 -8102.623,E2 -8102.623} C_VEL
LIN {X 0,Y 460.667,Z 257.915,A -85,B 0,C 180,E1 -8106.131,E2 -8106.131} C_VEL
LIN {X 0,Y 460.586,Z 257.924,A -85,B 0,C 180,E1 -8108.777,E2 -8108.777} C_VEL
LIN {X 0,Y 460.599,Z 257.924,A -85,B 0,C 180,E1 -8112.435,E2 -8112.435} C_VEL
LIN {X 0,Y 460.559,Z 257.928,A -85,B 0,C 180,E1 -8115.978,E2 -8115.978} C_VEL
LIN {X 0,Y 460.531,Z 257.931,A -85,B 0,C 180,E1 -8118.886,E2 -8118.886} C_VEL
LIN {X 0,Y 460.51,Z 257.935,A -85,B 0,C 180,E1 -8121.486,E2 -8121.486} C_VEL
LIN {X 0,Y 460.516,Z 257.933,A -85,B 0,C 180,E1 -8124.334,E2 -8124.334} C_VEL
LIN {X 0,Y 460.491,Z 257.938,A -85,B 0,C 180,E1 -8127.249,E2 -8127.249} C_VEL
LIN {X 0,Y 460.497,Z 257.936,A -85,B 0,C 180,E1 -8130.241,E2 -8130.241} C_VEL
LIN {X 0,Y 460.518,Z 257.934,A -85,B 0,C 180,E1 -8133.326,E2 -8133.326} C_VEL
LIN {X 0,Y 460.471,Z 257.939,A -85,B 0,C 180,E1 -8136.53,E2 -8136.53} C_VEL
LIN {X 0,Y 460.512,Z 257.935,A -85,B 0,C 180,E1 -8139.865,E2 -8139.865} C_VEL
LIN {X 0,Y 460.463,Z 257.941,A -85,B 0,C 180,E1 -8142.893,E2 -8142.893} C_VEL
LIN {X 0,Y 460.504,Z 257.935,A -85,B 0,C 180,E1 -8145.832,E2 -8145.832} C_VEL
LIN {X 0,Y 460.516,Z 257.934,A -85,B 0,C 180,E1 -8148.987,E2 -8148.987} C_VEL
LIN {X 0,Y 460.5,Z 257.936,A -85,B 0,C 180,E1 -8152.376,E2 -8152.376} C_VEL
LIN {X 0,Y 460.537,Z 257.931,A -85,B 0,C 180,E1 -8155.623,E2 -8155.623} C_VEL
LIN {X 0,Y 460.506,Z 257.935,A -85,B 0,C 180,E1 -8158.742,E2 -8158.742} C_VEL
LIN {X 0,Y 460.507,Z 257.934,A -85,B 0,C 180,E1 -8161.764,E2 -8161.764} C_VEL
LIN {X 0,Y 460.524,Z 257.933,A -85,B 0,C 180,E1 -8164.703,E2 -8164.703} C_VEL
LIN {X 0,Y 460.505,Z 257.934,A -85,B 0,C 180,E1 -8167.571,E2 -8167.571} C_VEL
LIN {X 0,Y 460.567,Z 257.931,A -85,B 0,C 180,E1 -8170.384,E2 -8170.384} C_VEL
LIN {X 0,Y 460.465,Z 257.94,A -85,B 0,C 180,E1 -8173.598,E2 -8173.598} C_VEL
LIN {X 0,Y 460.483,Z 258.076,A -85,B 0,C 180,E1 -8174.054,E2 -8174.054} C_VEL
LIN {X 0,Y 460.529,Z 267.456,A -85,B 0,C 180,E1 -8176.195,E2 -8176.195} C_VEL
LIN {X 0,Y 460.079,Z 268.935,A -85,B 0,C 180,E1 -8176.365,E2 -8176.365} C_VEL
LIN {X 0,Y 458.729,Z 271.657,A -85,B 0,C 180,E1 -8176.452,E2 -8176.452} C_VEL
LIN {X 0,Y 455.74,Z 278.998,A -85,B 0,C 180,E1 -8176.487,E2 -8176.487} C_VEL
LIN {X 0,Y 454.945,Z 283.154,A -85,B 0,C 180,E1 -8176.509,E2 -8176.509} C_VEL
LIN {X 0,Y 455.132,Z 289.717,A -85,B 0,C 180,E1 -8176.613,E2 -8176.613} C_VEL
LIN {X 0,Y 455.774,Z 298.51,A -85,B 0,C 180,E1 -8176.798,E2 -8176.798} C_VEL
LIN {X 0,Y 455.378,Z 345.158,A -85,B 0,C 180,E1 -8177.55,E2 -8177.55} C_VEL
LIN {X 0,Y 455.239,Z 354.258,A -85,B 0,C 180,E1 -8177.801,E2 -8177.801} C_VEL
LIN {X 0,Y 455.091,Z 363.838,A -85,B 0,C 180,E1 -8178.192,E2 -8178.192} C_VEL
LIN {X 0,Y 454.844,Z 373.861,A -85,B 0,C 180,E1 -8178.751,E2 -8178.751} C_VEL
LIN {X 0,Y 454.548,Z 384.254,A -85,B 0,C 180,E1 -8179.532,E2 -8179.532} C_VEL
LIN {X 0,Y 454.171,Z 392.377,A -85,B 0,C 180,E1 -8180.312,E2 -8180.312} C_VEL
LIN {X 0,Y 453.862,Z 399.074,A -85,B 0,C 180,E1 -8181.092,E2 -8181.092} C_VEL
LIN {X 0,Y 453.525,Z 405.412,A -85,B 0,C 180,E1 -8181.983,E2 -8181.983} C_VEL
LIN {X 0,Y 453.362,Z 410.672,A -85,B 0,C 180,E1 -8182.876,E2 -8182.876} C_VEL
LIN {X 0,Y 453.11,Z 415.069,A -85,B 0,C 180,E1 -8183.766,E2 -8183.766} C_VEL
LIN {X 0,Y 452.973,Z 418.726,A -85,B 0,C 180,E1 -8184.658,E2 -8184.658} C_VEL
LIN {X 0,Y 452.91,Z 421.707,A -85,B 0,C 180,E1 -8185.55,E2 -8185.55} C_VEL
LIN {X 0,Y 452.792,Z 424.019,A -85,B 0,C 180,E1 -8186.44,E2 -8186.44} C_VEL
LIN {X 0,Y 452.692,Z 425.782,A -85,B 0,C 180,E1 -8187.33,E2 -8187.33} C_VEL
LIN {X 0,Y 452.585,Z 427.056,A -85,B 0,C 180,E1 -8188.22,E2 -8188.22} C_VEL
LIN {X 0,Y 452.503,Z 427.864,A -85,B 0,C 180,E1 -8189.11,E2 -8189.11} C_VEL
LIN {X 0,Y 452.483,Z 428.17,A -85,B 0,C 180,E1 -8190,E2 -8190} C_VEL
LIN {X 0,Y 452.503,Z 427.897,A -85,B 0,C 180,E1 -8190.889,E2 -8190.889} C_VEL
LIN {X 0,Y 452.585,Z 427.157,A -85,B 0,C 180,E1 -8191.779,E2 -8191.779} C_VEL
LIN {X 0,Y 452.679,Z 425.952,A -85,B 0,C 180,E1 -8192.669,E2 -8192.669} C_VEL
LIN {X 0,Y 452.824,Z 423.12,A -85,B 0,C 180,E1 -8194.004,E2 -8194.004} C_VEL
LIN {X 0,Y 452.962,Z 420.542,A -85,B 0,C 180,E1 -8194.895,E2 -8194.895} C_VEL
LIN {X 0,Y 452.962,Z 417.367,A -85,B 0,C 180,E1 -8195.788,E2 -8195.788} C_VEL
LIN {X 0,Y 453.334,Z 412.473,A -85,B 0,C 180,E1 -8196.872,E2 -8196.872} C_VEL
LIN {X 0,Y 453.451,Z 407.553,A -85,B 0,C 180,E1 -8197.771,E2 -8197.771} C_VEL
LIN {X 0,Y 453.746,Z 401.47,A -85,B 0,C 180,E1 -8198.685,E2 -8198.685} C_VEL
LIN {X 0,Y 454.079,Z 394.235,A -85,B 0,C 180,E1 -8199.577,E2 -8199.577} C_VEL
LIN {X 0,Y 454.463,Z 386.496,A -85,B 0,C 180,E1 -8200.356,E2 -8200.356} C_VEL
LIN {X 0,Y 454.653,Z 378.34,A -85,B 0,C 180,E1 -8201.028,E2 -8201.028} C_VEL
LIN {X 0,Y 455.018,Z 369.814,A -85,B 0,C 180,E1 -8201.583,E2 -8201.583} C_VEL
LIN {X 0,Y 455.241,Z 358.547,A -85,B 0,C 180,E1 -8202.142,E2 -8202.142} C_VEL
LIN {X 0,Y 455.358,Z 347.306,A -85,B 0,C 180,E1 -8202.497,E2 -8202.497} C_VEL
LIN {X 0,Y 455.594,Z 326.991,A -85,B 0,C 180,E1 -8202.848,E2 -8202.848} C_VEL
LIN {X 0,Y 455.703,Z 280.659,A -85,B 0,C 180,E1 -8203.581,E2 -8203.581} C_VEL
LIN {X 0,Y 453.518,Z 269.008,A -85,B 0,C 180,E1 -8203.849,E2 -8203.849} C_VEL
LIN {X 0,Y 453.403,Z 258.861,A -85,B 0,C 180,E1 -8206.185,E2 -8206.185} C_VEL
LIN {X 0,Y 453.516,Z 258.807,A -85,B 0,C 180,E1 -8209.039,E2 -8209.039} C_VEL
LIN {X 0,Y 453.47,Z 258.811,A -85,B 0,C 180,E1 -8211.836,E2 -8211.836} C_VEL
LIN {X 0,Y 453.467,Z 258.812,A -85,B 0,C 180,E1 -8214.737,E2 -8214.737} C_VEL
LIN {X 0,Y 453.459,Z 258.813,A -85,B 0,C 180,E1 -8217.942,E2 -8217.942} C_VEL
LIN {X 0,Y 453.451,Z 258.816,A -85,B 0,C 180,E1 -8220.761,E2 -8220.761} C_VEL
LIN {X 0,Y 453.463,Z 258.812,A -85,B 0,C 180,E1 -8223.913,E2 -8223.913} C_VEL
LIN {X 0,Y 453.446,Z 258.814,A -85,B 0,C 180,E1 -8227.19,E2 -8227.19} C_VEL
LIN {X 0,Y 453.467,Z 258.814,A -85,B 0,C 180,E1 -8230.611,E2 -8230.611} C_VEL
LIN {X 0,Y 453.477,Z 258.812,A -85,B 0,C 180,E1 -8234.528,E2 -8234.528} C_VEL
LIN {X 0,Y 453.432,Z 258.816,A -85,B 0,C 180,E1 -8238.071,E2 -8238.071} C_VEL
LIN {X 0,Y 453.439,Z 258.815,A -85,B 0,C 180,E1 -8240.801,E2 -8240.801} C_VEL
LIN {X 0,Y 453.444,Z 258.814,A -85,B 0,C 180,E1 -8243.916,E2 -8243.916} C_VEL
LIN {X 0,Y 453.468,Z 258.813,A -85,B 0,C 180,E1 -8247.15,E2 -8247.15} C_VEL
LIN {X 0,Y 453.451,Z 258.814,A -85,B 0,C 180,E1 -8250.266,E2 -8250.266} C_VEL
LIN {X 0,Y 453.436,Z 258.815,A -85,B 0,C 180,E1 -8253.289,E2 -8253.289} C_VEL
LIN {X 0,Y 453.486,Z 258.809,A -85,B 0,C 180,E1 -8256.238,E2 -8256.238} C_VEL
LIN {X 0,Y 453.468,Z 258.811,A -85,B 0,C 180,E1 -8259.117,E2 -8259.117} C_VEL
LIN {X 0,Y 453.481,Z 258.81,A -85,B 0,C 180,E1 -8261.943,E2 -8261.943} C_VEL
LIN {X 0,Y 453.512,Z 258.807,A -85,B 0,C 180,E1 -8264.725,E2 -8264.725} C_VEL
LIN {X 0,Y 453.539,Z 258.804,A -85,B 0,C 180,E1 -8268.378,E2 -8268.378} C_VEL
LIN {X 0,Y 453.552,Z 258.8,A -85,B 0,C 180,E1 -8271.086,E2 -8271.086} C_VEL
LIN {X 0,Y 453.631,Z 258.791,A -85,B 0,C 180,E1 -8273.774,E2 -8273.774} C_VEL
LIN {X 0,Y 453.696,Z 258.783,A -85,B 0,C 180,E1 -8277.336,E2 -8277.336} C_VEL
LIN {X 0,Y 453.761,Z 258.776,A -85,B 0,C 180,E1 -8280,E2 -8280} C_VEL
LIN {X 0,Y 453.696,Z 258.782,A -85,B 0,C 180,E1 -8282.663,E2 -8282.663} C_VEL
LIN {X 0,Y 453.628,Z 258.793,A -85,B 0,C 180,E1 -8286.226,E2 -8286.226} C_VEL
LIN {X 0,Y 453.552,Z 258.8,A -85,B 0,C 180,E1 -8288.914,E2 -8288.914} C_VEL
LIN {X 0,Y 453.559,Z 258.799,A -85,B 0,C 180,E1 -8292.529,E2 -8292.529} C_VEL
LIN {X 0,Y 453.494,Z 258.808,A -85,B 0,C 180,E1 -8296.198,E2 -8296.198} C_VEL
LIN {X 0,Y 453.479,Z 258.809,A -85,B 0,C 180,E1 -8299.028,E2 -8299.028} C_VEL
LIN {X 0,Y 453.463,Z 258.814,A -85,B 0,C 180,E1 -8301.837,E2 -8301.837} C_VEL
LIN {X 0,Y 453.461,Z 258.811,A -85,B 0,C 180,E1 -8304.737,E2 -8304.737} C_VEL
LIN {X 0,Y 453.451,Z 258.813,A -85,B 0,C 180,E1 -8307.942,E2 -8307.942} C_VEL
LIN {X 0,Y 453.441,Z 258.813,A -85,B 0,C 180,E1 -8310.762,E2 -8310.762} C_VEL
LIN {X 0,Y 453.459,Z 258.811,A -85,B 0,C 180,E1 -8313.914,E2 -8313.914} C_VEL
LIN {X 0,Y 453.43,Z 258.819,A -85,B 0,C 180,E1 -8317.192,E2 -8317.192} C_VEL
LIN {X 0,Y 453.464,Z 258.81,A -85,B 0,C 180,E1 -8320.612,E2 -8320.612} C_VEL
LIN {X 0,Y 453.475,Z 258.809,A -85,B 0,C 180,E1 -8324.529,E2 -8324.529} C_VEL
LIN {X 0,Y 453.43,Z 258.813,A -85,B 0,C 180,E1 -8328.072,E2 -8328.072} C_VEL
LIN {X 0,Y 453.434,Z 258.818,A -85,B 0,C 180,E1 -8330.803,E2 -8330.803} C_VEL
LIN {X 0,Y 453.436,Z 258.812,A -85,B 0,C 180,E1 -8333.916,E2 -8333.916} C_VEL
LIN {X 0,Y 453.46,Z 258.816,A -85,B 0,C 180,E1 -8336.817,E2 -8336.817} C_VEL
LIN {X 0,Y 453.443,Z 258.813,A -85,B 0,C 180,E1 -8340.267,E2 -8340.267} C_VEL
LIN {X 0,Y 453.419,Z 258.818,A -85,B 0,C 180,E1 -8343.289,E2 -8343.289} C_VEL
LIN {X 0,Y 453.525,Z 258.947,A -85,B 0,C 180,E1 -8344.93,E2 -8344.93} C_VEL
LIN {X 0,Y 455.042,Z 268.036,A -85,B 0,C 180,E1 -8346.807,E2 -8346.807} C_VEL
LIN {X 0,Y 454.468,Z 282.599,A -85,B 0,C 180,E1 -8349.639,E2 -8349.639} C_VEL
LIN {X 0,Y 453.98,Z 295.896,A -85,B 0,C 180,E1 -8352.197,E2 -8352.197} C_VEL
LIN {X 0,Y 453.504,Z 311.551,A -85,B 0,C 180,E1 -8355.185,E2 -8355.185} C_VEL
LIN {X 0,Y 453.333,Z 317.086,A -85,B 0,C 180,E1 -8356.195,E2 -8356.195} C_VEL
LIN {X 0,Y 455.56,Z 336.503,A -85,B 0,C 180,E1 -8356.57,E2 -8356.57} C_VEL
LIN {X 0,Y 455.18,Z 394.379,A -85,B 0,C 180,E1 -8357.499,E2 -8357.499} C_VEL
LIN {X 0,Y 454.922,Z 403.971,A -85,B 0,C 180,E1 -8357.765,E2 -8357.765} C_VEL
LIN {X 0,Y 454.617,Z 414.04,A -85,B 0,C 180,E1 -8358.181,E2 -8358.181} C_VEL
LIN {X 0,Y 454.178,Z 425.483,A -85,B 0,C 180,E1 -8358.848,E2 -8358.848} C_VEL
LIN {X 0,Y 453.839,Z 434.099,A -85,B 0,C 180,E1 -8359.517,E2 -8359.517} C_VEL
LIN {X 0,Y 453.521,Z 442.209,A -85,B 0,C 180,E1 -8360.298,E2 -8360.298} C_VEL
LIN {X 0,Y 453.229,Z 448.912,A -85,B 0,C 180,E1 -8361.08,E2 -8361.08} C_VEL
LIN {X 0,Y 452.953,Z 455.277,A -85,B 0,C 180,E1 -8361.973,E2 -8361.973} C_VEL
LIN {X 0,Y 452.871,Z 460.577,A -85,B 0,C 180,E1 -8362.869,E2 -8362.869} C_VEL
LIN {X 0,Y 452.65,Z 464.99,A -85,B 0,C 180,E1 -8363.761,E2 -8363.761} C_VEL
LIN {X 0,Y 452.581,Z 470.204,A -85,B 0,C 180,E1 -8365.101,E2 -8365.101} C_VEL
LIN {X 0,Y 452.557,Z 474.034,A -85,B 0,C 180,E1 -8366.439,E2 -8366.439} C_VEL
LIN {X 0,Y 452.549,Z 475.796,A -85,B 0,C 180,E1 -8367.33,E2 -8367.33} C_VEL
LIN {X 0,Y 452.51,Z 477.057,A -85,B 0,C 180,E1 -8368.22,E2 -8368.22} C_VEL
LIN {X 0,Y 452.493,Z 477.842,A -85,B 0,C 180,E1 -8369.111,E2 -8369.111} C_VEL
LIN {X 0,Y 452.475,Z 478.138,A -85,B 0,C 180,E1 -8370,E2 -8370} C_VEL
LIN {X 0,Y 452.493,Z 477.84,A -85,B 0,C 180,E1 -8370.89,E2 -8370.89} C_VEL
LIN {X 0,Y 452.51,Z 477.053,A -85,B 0,C 180,E1 -8371.78,E2 -8371.78} C_VEL
LIN {X 0,Y 452.55,Z 475.79,A -85,B 0,C 180,E1 -8372.671,E2 -8372.671} C_VEL
LIN {X 0,Y 452.524,Z 472.859,A -85,B 0,C 180,E1 -8374.008,E2 -8374.008} C_VEL
LIN {X 0,Y 452.582,Z 470.193,A -85,B 0,C 180,E1 -8374.9,E2 -8374.9} C_VEL
LIN {X 0,Y 452.65,Z 464.974,A -85,B 0,C 180,E1 -8376.24,E2 -8376.24} C_VEL
LIN {X 0,Y 452.881,Z 458.106,A -85,B 0,C 180,E1 -8377.58,E2 -8377.58} C_VEL
LIN {X 0,Y 453.13,Z 450.602,A -85,B 0,C 180,E1 -8378.698,E2 -8378.698} C_VEL
LIN {X 0,Y 453.462,Z 443.21,A -85,B 0,C 180,E1 -8379.591,E2 -8379.591} C_VEL
LIN {X 0,Y 453.794,Z 435.299,A -85,B 0,C 180,E1 -8380.372,E2 -8380.372} C_VEL
LIN {X 0,Y 454.114,Z 426.943,A -85,B 0,C 180,E1 -8381.042,E2 -8381.042} C_VEL
LIN {X 0,Y 454.584,Z 416.286,A -85,B 0,C 180,E1 -8381.708,E2 -8381.708} C_VEL
LIN {X 0,Y 454.895,Z 405.531,A -85,B 0,C 180,E1 -8382.181,E2 -8382.181} C_VEL
LIN {X 0,Y 455.182,Z 395.015,A -85,B 0,C 180,E1 -8382.484,E2 -8382.484} C_VEL
LIN {X 0,Y 455.573,Z 342.162,A -85,B 0,C 180,E1 -8383.337,E2 -8383.337} C_VEL
LIN {X 0,Y 455.287,Z 334.296,A -85,B 0,C 180,E1 -8383.47,E2 -8383.47} C_VEL
LIN {X 0,Y 453.306,Z 316.83,A -85,B 0,C 180,E1 -8383.811,E2 -8383.811} C_VEL
LIN {X 0,Y 453.766,Z 301.901,A -85,B 0,C 180,E1 -8386.651,E2 -8386.651} C_VEL
LIN {X 0,Y 454.355,Z 286.808,A -85,B 0,C 180,E1 -8389.543,E2 -8389.543} C_VEL
LIN {X 0,Y 454.988,Z 270.441,A -85,B 0,C 180,E1 -8392.716,E2 -8392.716} C_VEL
LIN {X 0,Y 454.907,Z 266.78,A -85,B 0,C 180,E1 -8393.442,E2 -8393.442} C_VEL
LIN {X 0,Y 453.504,Z 258.809,A -85,B 0,C 180,E1 -8395.102,E2 -8395.102} C_VEL
LIN {X 0,Y 453.447,Z 258.812,A -85,B 0,C 180,E1 -8398.716,E2 -8398.716} C_VEL
LIN {X 0,Y 453.434,Z 258.814,A -85,B 0,C 180,E1 -8401.802,E2 -8401.802} C_VEL
LIN {X 0,Y 453.466,Z 258.813,A -85,B 0,C 180,E1 -8404.991,E2 -8404.991} C_VEL
LIN {X 0,Y 453.438,Z 258.812,A -85,B 0,C 180,E1 -8408.315,E2 -8408.315} C_VEL
LIN {X 0,Y 453.464,Z 258.811,A -85,B 0,C 180,E1 -8410.613,E2 -8410.613} C_VEL
LIN {X 0,Y 453.48,Z 258.809,A -85,B 0,C 180,E1 -8414.528,E2 -8414.528} C_VEL
LIN {X 0,Y 453.433,Z 258.813,A -85,B 0,C 180,E1 -8418.072,E2 -8418.072} C_VEL
LIN {X 0,Y 453.429,Z 258.82,A -85,B 0,C 180,E1 -8420.804,E2 -8420.804} C_VEL
LIN {X 0,Y 453.44,Z 258.813,A -85,B 0,C 180,E1 -8423.916,E2 -8423.916} C_VEL
LIN {X 0,Y 453.465,Z 258.813,A -85,B 0,C 180,E1 -8426.816,E2 -8426.816} C_VEL
LIN {X 0,Y 453.447,Z 258.814,A -85,B 0,C 180,E1 -8430.266,E2 -8430.266} C_VEL
LIN {X 0,Y 453.423,Z 258.816,A -85,B 0,C 180,E1 -8433.289,E2 -8433.289} C_VEL
LIN {X 0,Y 453.47,Z 258.813,A -85,B 0,C 180,E1 -8436.237,E2 -8436.237} C_VEL
LIN {X 0,Y 453.437,Z 258.814,A -85,B 0,C 180,E1 -8439.116,E2 -8439.116} C_VEL
LIN {X 0,Y 453.456,Z 258.813,A -85,B 0,C 180,E1 -8441.942,E2 -8441.942} C_VEL
LIN {X 0,Y 453.485,Z 258.809,A -85,B 0,C 180,E1 -8444.725,E2 -8444.725} C_VEL
LIN {X 0,Y 453.566,Z 258.798,A -85,B 0,C 180,E1 -8447.471,E2 -8447.471} C_VEL
LIN {X 0,Y 453.556,Z 258.8,A -85,B 0,C 180,E1 -8451.086,E2 -8451.086} C_VEL
LIN {X 0,Y 453.635,Z 258.792,A -85,B 0,C 180,E1 -8453.774,E2 -8453.774} C_VEL
LIN {X 0,Y 453.702,Z 258.781,A -85,B 0,C 180,E1 -8457.337,E2 -8457.337} C_VEL
LIN {X 0,Y 453.768,Z 258.775,A -85,B 0,C 180,E1 -8460,E2 -8460} C_VEL
LIN {X 0,Y 453.702,Z 258.783,A -85,B 0,C 180,E1 -8462.664,E2 -8462.664} C_VEL
LIN {X 0,Y 453.635,Z 258.79,A -85,B 0,C 180,E1 -8466.226,E2 -8466.226} C_VEL
LIN {X 0,Y 453.556,Z 258.8,A -85,B 0,C 180,E1 -8468.914,E2 -8468.914} C_VEL
LIN {X 0,Y 453.566,Z 258.799,A -85,B 0,C 180,E1 -8472.529,E2 -8472.529} C_VEL
LIN {X 0,Y 453.498,Z 258.808,A -85,B 0,C 180,E1 -8476.198,E2 -8476.198} C_VEL
LIN {X 0,Y 453.487,Z 258.809,A -85,B 0,C 180,E1 -8479.027,E2 -8479.027} C_VEL
LIN {X 0,Y 453.47,Z 258.811,A -85,B 0,C 180,E1 -8481.837,E2 -8481.837} C_VEL
LIN {X 0,Y 453.469,Z 258.811,A -85,B 0,C 180,E1 -8484.737,E2 -8484.737} C_VEL
LIN {X 0,Y 453.461,Z 258.813,A -85,B 0,C 180,E1 -8487.942,E2 -8487.942} C_VEL
LIN {X 0,Y 453.455,Z 258.813,A -85,B 0,C 180,E1 -8490.761,E2 -8490.761} C_VEL
LIN {X 0,Y 453.467,Z 258.813,A -85,B 0,C 180,E1 -8493.914,E2 -8493.914} C_VEL
LIN {X 0,Y 453.448,Z 258.814,A -85,B 0,C 180,E1 -8497.19,E2 -8497.19} C_VEL
LIN {X 0,Y 453.471,Z 258.811,A -85,B 0,C 180,E1 -8500.612,E2 -8500.612} C_VEL
LIN {X 0,Y 453.482,Z 258.81,A -85,B 0,C 180,E1 -8504.528,E2 -8504.528} C_VEL
LIN {X 0,Y 453.437,Z 258.815,A -85,B 0,C 180,E1 -8508.071,E2 -8508.071} C_VEL
LIN {X 0,Y 453.449,Z 258.814,A -85,B 0,C 180,E1 -8510.801,E2 -8510.801} C_VEL
LIN {X 0,Y 453.452,Z 258.813,A -85,B 0,C 180,E1 -8513.917,E2 -8513.917} C_VEL
LIN {X 0,Y 453.474,Z 258.812,A -85,B 0,C 180,E1 -8517.15,E2 -8517.15} C_VEL
LIN {X 0,Y 453.456,Z 258.813,A -85,B 0,C 180,E1 -8520.267,E2 -8520.267} C_VEL
LIN {X 0,Y 453.444,Z 258.816,A -85,B 0,C 180,E1 -8523.29,E2 -8523.29} C_VEL
LIN {X 0,Y 453.494,Z 258.808,A -85,B 0,C 180,E1 -8526.238,E2 -8526.238} C_VEL
LIN {X 0,Y 453.482,Z 258.811,A -85,B 0,C 180,E1 -8529.117,E2 -8529.117} C_VEL
LIN {X 0,Y 453.486,Z 258.809,A -85,B 0,C 180,E1 -8531.943,E2 -8531.943} C_VEL
LIN {X 0,Y 453.446,Z 258.954,A -85,B 0,C 180,E1 -8533.934,E2 -8533.934} C_VEL
LIN {X 0,Y 453.516,Z 269.041,A -85,B 0,C 180,E1 -8536.254,E2 -8536.254} C_VEL
LIN {X 0,Y 455.914,Z 281.889,A -85,B 0,C 180,E1 -8536.539,E2 -8536.539} C_VEL
LIN {X 0,Y 455.774,Z 298.51,A -85,B 0,C 180,E1 -8536.798,E2 -8536.798} C_VEL
LIN {X 0,Y 455.03,Z 304.35,A -85,B 0,C 180,E1 -8536.869,E2 -8536.869} C_VEL
LIN {X 0,Y 449.361,Z 323.331,A -85,B 0,C 180,E1 -8537,E2 -8537} C_VEL
LIN {X 0,Y 448.631,Z 329.171,A -85,B 0,C 180,E1 -8537.072,E2 -8537.072} C_VEL
LIN {X 0,Y 448.443,Z 346.864,A -85,B 0,C 180,E1 -8537.383,E2 -8537.383} C_VEL
LIN {X 0,Y 448.286,Z 357.974,A -85,B 0,C 180,E1 -8537.723,E2 -8537.723} C_VEL
LIN {X 0,Y 448.06,Z 368.664,A -85,B 0,C 180,E1 -8538.234,E2 -8538.234} C_VEL
LIN {X 0,Y 447.763,Z 377.491,A -85,B 0,C 180,E1 -8538.8,E2 -8538.8} C_VEL
LIN {X 0,Y 447.502,Z 385.875,A -85,B 0,C 180,E1 -8539.48,E2 -8539.48} C_VEL
LIN {X 0,Y 447.141,Z 393.787,A -85,B 0,C 180,E1 -8540.272,E2 -8540.272} C_VEL
LIN {X 0,Y 446.858,Z 399.468,A -85,B 0,C 180,E1 -8540.951,E2 -8540.951} C_VEL
LIN {X 0,Y 446.527,Z 405.805,A -85,B 0,C 180,E1 -8541.856,E2 -8541.856} C_VEL
LIN {X 0,Y 446.321,Z 411.066,A -85,B 0,C 180,E1 -8542.763,E2 -8542.763} C_VEL
LIN {X 0,Y 446.088,Z 415.461,A -85,B 0,C 180,E1 -8543.668,E2 -8543.668} C_VEL
LIN {X 0,Y 445.903,Z 419.12,A -85,B 0,C 180,E1 -8544.573,E2 -8544.573} C_VEL
LIN {X 0,Y 445.853,Z 422.099,A -85,B 0,C 180,E1 -8545.479,E2 -8545.479} C_VEL
LIN {X 0,Y 445.729,Z 424.411,A -85,B 0,C 180,E1 -8546.384,E2 -8546.384} C_VEL
LIN {X 0,Y 445.614,Z 426.174,A -85,B 0,C 180,E1 -8547.288,E2 -8547.288} C_VEL
LIN {X 0,Y 445.512,Z 427.448,A -85,B 0,C 180,E1 -8548.192,E2 -8548.192} C_VEL
LIN {X 0,Y 445.44,Z 428.254,A -85,B 0,C 180,E1 -8549.096,E2 -8549.096} C_VEL
LIN {X 0,Y 445.418,Z 428.561,A -85,B 0,C 180,E1 -8550,E2 -8550} C_VEL
LIN {X 0,Y 445.441,Z 428.287,A -85,B 0,C 180,E1 -8550.904,E2 -8550.904} C_VEL
LIN {X 0,Y 445.511,Z 427.548,A -85,B 0,C 180,E1 -8551.808,E2 -8551.808} C_VEL
LIN {X 0,Y 445.602,Z 426.343,A -85,B 0,C 180,E1 -8552.712,E2 -8552.712} C_VEL
LIN {X 0,Y 445.767,Z 423.509,A -85,B 0,C 180,E1 -8554.068,E2 -8554.068} C_VEL
LIN {X 0,Y 445.907,Z 420.931,A -85,B 0,C 180,E1 -8554.972,E2 -8554.972} C_VEL
LIN {X 0,Y 445.92,Z 417.756,A -85,B 0,C 180,E1 -8555.879,E2 -8555.879} C_VEL
LIN {X 0,Y 446.296,Z 413.199,A -85,B 0,C 180,E1 -8556.915,E2 -8556.915} C_VEL
LIN {X 0,Y 446.443,Z 407.8,A -85,B 0,C 180,E1 -8557.917,E2 -8557.917} C_VEL
LIN {X 0,Y 446.757,Z 401.858,A -85,B 0,C 180,E1 -8558.822,E2 -8558.822} C_VEL
LIN {X 0,Y 447.11,Z 394.621,A -85,B 0,C 180,E1 -8559.728,E2 -8559.728} C_VEL
LIN {X 0,Y 447.511,Z 386.881,A -85,B 0,C 180,E1 -8560.519,E2 -8560.519} C_VEL
LIN {X 0,Y 447.707,Z 378.725,A -85,B 0,C 180,E1 -8561.201,E2 -8561.201} C_VEL
LIN {X 0,Y 448.085,Z 370.197,A -85,B 0,C 180,E1 -8561.765,E2 -8561.765} C_VEL
LIN {X 0,Y 448.329,Z 358.926,A -85,B 0,C 180,E1 -8562.332,E2 -8562.332} C_VEL
LIN {X 0,Y 448.453,Z 347.703,A -85,B 0,C 180,E1 -8562.692,E2 -8562.692} C_VEL
LIN {X 0,Y 448.736,Z 325.775,A -85,B 0,C 180,E1 -8563.073,E2 -8563.073} C_VEL
LIN {X 0,Y 448.853,Z 281.77,A -85,B 0,C 180,E1 -8563.78,E2 -8563.78} C_VEL
LIN {X 0,Y 446.53,Z 269.409,A -85,B 0,C 180,E1 -8564.062,E2 -8564.062} C_VEL
LIN {X 0,Y 446.403,Z 260.036,A -85,B 0,C 180,E1 -8566.239,E2 -8566.239} C_VEL
LIN {X 0,Y 446.36,Z 259.702,A -85,B 0,C 180,E1 -8566.324,E2 -8566.324} C_VEL
LIN {X 0,Y 446.467,Z 259.689,A -85,B 0,C 180,E1 -8569.303,E2 -8569.303} C_VEL
LIN {X 0,Y 446.408,Z 259.69,A -85,B 0,C 180,E1 -8572.2,E2 -8572.2} C_VEL
LIN {X 0,Y 446.419,Z 259.691,A -85,B 0,C 180,E1 -8575.154,E2 -8575.154} C_VEL
LIN {X 0,Y 446.414,Z 259.69,A -85,B 0,C 180,E1 -8578.183,E2 -8578.183} C_VEL
LIN {X 0,Y 446.39,Z 259.693,A -85,B 0,C 180,E1 -8581.302,E2 -8581.302} C_VEL
LIN {X 0,Y 446.419,Z 259.691,A -85,B 0,C 180,E1 -8584.523,E2 -8584.523} C_VEL
LIN {X 0,Y 446.407,Z 259.691,A -85,B 0,C 180,E1 -8588.078,E2 -8588.078} C_VEL
LIN {X 0,Y 446.397,Z 259.693,A -85,B 0,C 180,E1 -8591.394,E2 -8591.394} C_VEL
LIN {X 0,Y 446.417,Z 259.69,A -85,B 0,C 180,E1 -8595.107,E2 -8595.107} C_VEL
LIN {X 0,Y 446.396,Z 259.693,A -85,B 0,C 180,E1 -8598.605,E2 -8598.605} C_VEL
LIN {X 0,Y 446.402,Z 259.692,A -85,B 0,C 180,E1 -8601.922,E2 -8601.922} C_VEL
LIN {X 0,Y 446.416,Z 259.69,A -85,B 0,C 180,E1 -8605.476,E2 -8605.476} C_VEL
LIN {X 0,Y 446.402,Z 259.692,A -85,B 0,C 180,E1 -8608.698,E2 -8608.698} C_VEL
LIN {X 0,Y 446.418,Z 259.69,A -85,B 0,C 180,E1 -8611.836,E2 -8611.836} C_VEL
LIN {X 0,Y 446.416,Z 259.692,A -85,B 0,C 180,E1 -8614.845,E2 -8614.845} C_VEL
LIN {X 0,Y 446.441,Z 259.687,A -85,B 0,C 180,E1 -8618.246,E2 -8618.246} C_VEL
LIN {X 0,Y 446.435,Z 259.688,A -85,B 0,C 180,E1 -8621.648,E2 -8621.648} C_VEL
LIN {X 0,Y 446.453,Z 259.686,A -85,B 0,C 180,E1 -8624.478,E2 -8624.478} C_VEL
LIN {X 0,Y 446.511,Z 259.678,A -85,B 0,C 180,E1 -8627.384,E2 -8627.384} C_VEL
LIN {X 0,Y 446.503,Z 259.679,A -85,B 0,C 180,E1 -8630.944,E2 -8630.944} C_VEL
LIN {X 0,Y 446.601,Z 259.667,A -85,B 0,C 180,E1 -8633.676,E2 -8633.676} C_VEL
LIN {X 0,Y 446.646,Z 259.661,A -85,B 0,C 180,E1 -8637.294,E2 -8637.294} C_VEL
LIN {X 0,Y 446.712,Z 259.654,A -85,B 0,C 180,E1 -8640,E2 -8640} C_VEL
LIN {X 0,Y 446.645,Z 259.661,A -85,B 0,C 180,E1 -8642.706,E2 -8642.706} C_VEL
LIN {X 0,Y 446.598,Z 259.668,A -85,B 0,C 180,E1 -8646.324,E2 -8646.324} C_VEL
LIN {X 0,Y 446.502,Z 259.679,A -85,B 0,C 180,E1 -8649.056,E2 -8649.056} C_VEL
LIN {X 0,Y 446.516,Z 259.676,A -85,B 0,C 180,E1 -8652.73,E2 -8652.73} C_VEL
LIN {X 0,Y 446.448,Z 259.686,A -85,B 0,C 180,E1 -8656.209,E2 -8656.209} C_VEL
LIN {X 0,Y 446.425,Z 259.688,A -85,B 0,C 180,E1 -8659.305,E2 -8659.305} C_VEL
LIN {X 0,Y 446.401,Z 259.691,A -85,B 0,C 180,E1 -8662.2,E2 -8662.2} C_VEL
LIN {X 0,Y 446.414,Z 259.69,A -85,B 0,C 180,E1 -8665.155,E2 -8665.155} C_VEL
LIN {X 0,Y 446.409,Z 259.689,A -85,B 0,C 180,E1 -8668.184,E2 -8668.184} C_VEL
LIN {X 0,Y 446.385,Z 259.696,A -85,B 0,C 180,E1 -8671.303,E2 -8671.303} C_VEL
LIN {X 0,Y 446.414,Z 259.688,A -85,B 0,C 180,E1 -8674.524,E2 -8674.524} C_VEL
LIN {X 0,Y 446.392,Z 259.691,A -85,B 0,C 180,E1 -8678.076,E2 -8678.076} C_VEL
LIN {X 0,Y 446.395,Z 259.694,A -85,B 0,C 180,E1 -8681.395,E2 -8681.395} C_VEL
LIN {X 0,Y 446.444,Z 259.69,A -85,B 0,C 180,E1 -8685.105,E2 -8685.105} C_VEL
LIN {X 0,Y 446.395,Z 259.692,A -85,B 0,C 180,E1 -8688.606,E2 -8688.606} C_VEL
LIN {X 0,Y 446.393,Z 259.69,A -85,B 0,C 180,E1 -8691.924,E2 -8691.924} C_VEL
LIN {X 0,Y 446.409,Z 259.688,A -85,B 0,C 180,E1 -8695.476,E2 -8695.476} C_VEL
LIN {X 0,Y 446.384,Z 259.697,A -85,B 0,C 180,E1 -8698.698,E2 -8698.698} C_VEL
LIN {X 0,Y 446.397,Z 259.691,A -85,B 0,C 180,E1 -8701.843,E2 -8701.843} C_VEL
LIN {X 0,Y 446.474,Z 259.764,A -85,B 0,C 180,E1 -8704.756,E2 -8704.756} C_VEL
LIN {X 0,Y 448.053,Z 268.856,A -85,B 0,C 180,E1 -8706.668,E2 -8706.668} C_VEL
LIN {X 0,Y 447.499,Z 282.204,A -85,B 0,C 180,E1 -8709.307,E2 -8709.307} C_VEL
LIN {X 0,Y 446.992,Z 295.502,A -85,B 0,C 180,E1 -8711.91,E2 -8711.91} C_VEL
LIN {X 0,Y 446.492,Z 311.157,A -85,B 0,C 180,E1 -8714.947,E2 -8714.947} C_VEL
LIN {X 0,Y 446.29,Z 316.461,A -85,B 0,C 180,E1 -8715.969,E2 -8715.969} C_VEL
LIN {X 0,Y 448.681,Z 337.724,A -85,B 0,C 180,E1 -8716.386,E2 -8716.386} C_VEL
LIN {X 0,Y 448.266,Z 394.036,A -85,B 0,C 180,E1 -8717.304,E2 -8717.304} C_VEL
LIN {X 0,Y 448,Z 403.588,A -85,B 0,C 180,E1 -8717.573,E2 -8717.573} C_VEL
LIN {X 0,Y 447.664,Z 413.653,A -85,B 0,C 180,E1 -8717.994,E2 -8717.994} C_VEL
LIN {X 0,Y 447.209,Z 425.095,A -85,B 0,C 180,E1 -8718.672,E2 -8718.672} C_VEL
LIN {X 0,Y 446.837,Z 433.708,A -85,B 0,C 180,E1 -8719.351,E2 -8719.351} C_VEL
LIN {X 0,Y 446.496,Z 441.818,A -85,B 0,C 180,E1 -8720.144,E2 -8720.144} C_VEL
LIN {X 0,Y 446.2,Z 448.521,A -85,B 0,C 180,E1 -8720.938,E2 -8720.938} C_VEL
LIN {X 0,Y 445.904,Z 454.886,A -85,B 0,C 180,E1 -8721.846,E2 -8721.846} C_VEL
LIN {X 0,Y 445.785,Z 460.184,A -85,B 0,C 180,E1 -8722.755,E2 -8722.755} C_VEL
LIN {X 0,Y 445.576,Z 464.598,A -85,B 0,C 180,E1 -8723.662,E2 -8723.662} C_VEL
LIN {X 0,Y 445.511,Z 469.813,A -85,B 0,C 180,E1 -8725.023,E2 -8725.023} C_VEL
LIN {X 0,Y 445.454,Z 473.641,A -85,B 0,C 180,E1 -8726.382,E2 -8726.382} C_VEL
LIN {X 0,Y 445.474,Z 475.406,A -85,B 0,C 180,E1 -8727.288,E2 -8727.288} C_VEL
LIN {X 0,Y 445.425,Z 476.666,A -85,B 0,C 180,E1 -8728.192,E2 -8728.192} C_VEL
LIN {X 0,Y 445.43,Z 477.452,A -85,B 0,C 180,E1 -8729.096,E2 -8729.096} C_VEL
LIN {X 0,Y 445.411,Z 477.748,A -85,B 0,C 180,E1 -8730,E2 -8730} C_VEL
LIN {X 0,Y 445.43,Z 477.45,A -85,B 0,C 180,E1 -8730.905,E2 -8730.905} C_VEL
LIN {X 0,Y 445.425,Z 476.661,A -85,B 0,C 180,E1 -8731.809,E2 -8731.809} C_VEL
LIN {X 0,Y 445.474,Z 475.398,A -85,B 0,C 180,E1 -8732.713,E2 -8732.713} C_VEL
LIN {X 0,Y 445.428,Z 472.466,A -85,B 0,C 180,E1 -8734.072,E2 -8734.072} C_VEL
LIN {X 0,Y 445.512,Z 469.8,A -85,B 0,C 180,E1 -8734.978,E2 -8734.978} C_VEL
LIN {X 0,Y 445.576,Z 464.145,A -85,B 0,C 180,E1 -8736.441,E2 -8736.441} C_VEL
LIN {X 0,Y 445.816,Z 457.711,A -85,B 0,C 180,E1 -8737.701,E2 -8737.701} C_VEL
LIN {X 0,Y 446.097,Z 450.207,A -85,B 0,C 180,E1 -8738.836,E2 -8738.836} C_VEL
LIN {X 0,Y 446.449,Z 442.815,A -85,B 0,C 180,E1 -8739.743,E2 -8739.743} C_VEL
LIN {X 0,Y 446.784,Z 434.902,A -85,B 0,C 180,E1 -8740.537,E2 -8740.537} C_VEL
LIN {X 0,Y 447.142,Z 426.547,A -85,B 0,C 180,E1 -8741.216,E2 -8741.216} C_VEL
LIN {X 0,Y 447.629,Z 415.889,A -85,B 0,C 180,E1 -8741.892,E2 -8741.892} C_VEL
LIN {X 0,Y 447.978,Z 404.298,A -85,B 0,C 180,E1 -8742.4,E2 -8742.4} C_VEL
LIN {X 0,Y 448.231,Z 394.609,A -85,B 0,C 180,E1 -8742.681,E2 -8742.681} C_VEL
LIN {X 0,Y 448.567,Z 357.744,A -85,B 0,C 180,E1 -8743.292,E2 -8743.292} C_VEL
LIN {X 0,Y 448.487,Z 336.126,A -85,B 0,C 180,E1 -8743.642,E2 -8743.642} C_VEL
LIN {X 0,Y 446.31,Z 316.325,A -85,B 0,C 180,E1 -8744.052,E2 -8744.052} C_VEL
LIN {X 0,Y 446.887,Z 297.887,A -85,B 0,C 180,E1 -8747.622,E2 -8747.622} C_VEL
LIN {X 0,Y 447.422,Z 284.598,A -85,B 0,C 180,E1 -8750.217,E2 -8750.217} C_VEL
LIN {X 0,Y 448.072,Z 270.044,A -85,B 0,C 180,E1 -8753.087,E2 -8753.087} C_VEL
LIN {X 0,Y 446.971,Z 262.486,A -85,B 0,C 180,E1 -8754.661,E2 -8754.661} C_VEL
LIN {X 0,Y 446.455,Z 259.687,A -85,B 0,C 180,E1 -8755.277,E2 -8755.277} C_VEL
LIN {X 0,Y 446.415,Z 259.687,A -85,B 0,C 180,E1 -8758.184,E2 -8758.184} C_VEL
LIN {X 0,Y 446.388,Z 259.697,A -85,B 0,C 180,E1 -8761.303,E2 -8761.303} C_VEL
LIN {X 0,Y 446.411,Z 259.688,A -85,B 0,C 180,E1 -8764.525,E2 -8764.525} C_VEL
LIN {X 0,Y 446.386,Z 259.691,A -85,B 0,C 180,E1 -8767.881,E2 -8767.881} C_VEL
LIN {X 0,Y 446.394,Z 259.692,A -85,B 0,C 180,E1 -8771.395,E2 -8771.395} C_VEL
LIN {X 0,Y 446.449,Z 259.687,A -85,B 0,C 180,E1 -8775.104,E2 -8775.104} C_VEL
LIN {X 0,Y 446.397,Z 259.693,A -85,B 0,C 180,E1 -8778.606,E2 -8778.606} C_VEL
LIN {X 0,Y 446.394,Z 259.69,A -85,B 0,C 180,E1 -8781.925,E2 -8781.925} C_VEL
LIN {X 0,Y 446.413,Z 259.688,A -85,B 0,C 180,E1 -8785.476,E2 -8785.476} C_VEL
LIN {X 0,Y 446.388,Z 259.695,A -85,B 0,C 180,E1 -8788.698,E2 -8788.698} C_VEL
LIN {X 0,Y 446.4,Z 259.69,A -85,B 0,C 180,E1 -8791.842,E2 -8791.842} C_VEL
LIN {X 0,Y 446.406,Z 259.691,A -85,B 0,C 180,E1 -8794.845,E2 -8794.845} C_VEL
LIN {X 0,Y 446.443,Z 259.689,A -85,B 0,C 180,E1 -8798.248,E2 -8798.248} C_VEL
LIN {X 0,Y 446.41,Z 259.689,A -85,B 0,C 180,E1 -8801.647,E2 -8801.647} C_VEL
LIN {X 0,Y 446.428,Z 259.689,A -85,B 0,C 180,E1 -8804.477,E2 -8804.477} C_VEL
LIN {X 0,Y 446.517,Z 259.676,A -85,B 0,C 180,E1 -8807.385,E2 -8807.385} C_VEL
LIN {X 0,Y 446.507,Z 259.678,A -85,B 0,C 180,E1 -8810.944,E2 -8810.944} C_VEL
LIN {X 0,Y 446.605,Z 259.667,A -85,B 0,C 180,E1 -8813.676,E2 -8813.676} C_VEL
LIN {X 0,Y 446.651,Z 259.66,A -85,B 0,C 180,E1 -8817.294,E2 -8817.294} C_VEL
LIN {X 0,Y 446.718,Z 259.653,A -85,B 0,C 180,E1 -8820,E2 -8820} C_VEL
LIN {X 0,Y 446.651,Z 259.661,A -85,B 0,C 180,E1 -8822.706,E2 -8822.706} C_VEL
LIN {X 0,Y 446.606,Z 259.666,A -85,B 0,C 180,E1 -8826.324,E2 -8826.324} C_VEL
LIN {X 0,Y 446.507,Z 259.678,A -85,B 0,C 180,E1 -8829.056,E2 -8829.056} C_VEL
LIN {X 0,Y 446.523,Z 259.676,A -85,B 0,C 180,E1 -8832.73,E2 -8832.73} C_VEL
LIN {X 0,Y 446.451,Z 259.686,A -85,B 0,C 180,E1 -8836.207,E2 -8836.207} C_VEL
LIN {X 0,Y 446.433,Z 259.69,A -85,B 0,C 180,E1 -8839.305,E2 -8839.305} C_VEL
LIN {X 0,Y 446.408,Z 259.692,A -85,B 0,C 180,E1 -8842.2,E2 -8842.2} C_VEL
LIN {X 0,Y 446.422,Z 259.691,A -85,B 0,C 180,E1 -8845.155,E2 -8845.155} C_VEL
LIN {X 0,Y 446.417,Z 259.69,A -85,B 0,C 180,E1 -8848.183,E2 -8848.183} C_VEL
LIN {X 0,Y 446.408,Z 259.691,A -85,B 0,C 180,E1 -8851.301,E2 -8851.301} C_VEL
LIN {X 0,Y 446.422,Z 259.689,A -85,B 0,C 180,E1 -8854.524,E2 -8854.524} C_VEL
LIN {X 0,Y 446.408,Z 259.691,A -85,B 0,C 180,E1 -8858.078,E2 -8858.078} C_VEL
LIN {X 0,Y 446.401,Z 259.692,A -85,B 0,C 180,E1 -8861.394,E2 -8861.394} C_VEL
LIN {X 0,Y 446.423,Z 259.689,A -85,B 0,C 180,E1 -8865.108,E2 -8865.108} C_VEL
LIN {X 0,Y 446.401,Z 259.693,A -85,B 0,C 180,E1 -8868.606,E2 -8868.606} C_VEL
LIN {X 0,Y 446.412,Z 259.69,A -85,B 0,C 180,E1 -8871.922,E2 -8871.922} C_VEL
LIN {X 0,Y 446.423,Z 259.691,A -85,B 0,C 180,E1 -8875.476,E2 -8875.476} C_VEL
LIN {X 0,Y 446.394,Z 259.692,A -85,B 0,C 180,E1 -8878.698,E2 -8878.698} C_VEL
LIN {X 0,Y 446.425,Z 259.688,A -85,B 0,C 180,E1 -8881.836,E2 -8881.836} C_VEL
LIN {X 0,Y 446.432,Z 259.688,A -85,B 0,C 180,E1 -8884.846,E2 -8884.846} C_VEL
LIN {X 0,Y 446.449,Z 259.685,A -85,B 0,C 180,E1 -8888.245,E2 -8888.245} C_VEL
LIN {X 0,Y 446.441,Z 259.686,A -85,B 0,C 180,E1 -8891.648,E2 -8891.648} C_VEL
LIN {X 0,Y 446.409,Z 259.845,A -85,B 0,C 180,E1 -8893.811,E2 -8893.811} C_VEL
LIN {X 0,Y 446.56,Z 269.31,A -85,B 0,C 180,E1 -8896.013,E2 -8896.013} C_VEL
LIN {X 0,Y 448.985,Z 282.31,A -85,B 0,C 180,E1 -8896.327,E2 -8896.327} C_VEL
LIN {X 0,Y 448.631,Z 329.171,A -85,B 0,C 180,E1 -8897.072,E2 -8897.072} C_VEL
LIN {X 0,Y 447.862,Z 335.018,A -85,B 0,C 180,E1 -8897.141,E2 -8897.141} C_VEL
LIN {X 0,Y 443.003,Z 350.086,A -85,B 0,C 180,E1 -8897.292,E2 -8897.292} C_VEL
LIN {X 0,Y 441.457,Z 357.623,A -85,B 0,C 180,E1 -8897.502,E2 -8897.502} C_VEL
LIN {X 0,Y 441.38,Z 359.502,A -85,B 0,C 180,E1 -8897.574,E2 -8897.574} C_VEL
LIN {X 0,Y 441.144,Z 369.061,A -85,B 0,C 180,E1 -8898.047,E2 -8898.047} C_VEL
LIN {X 0,Y 440.765,Z 379.382,A -85,B 0,C 180,E1 -8898.736,E2 -8898.736} C_VEL
LIN {X 0,Y 440.553,Z 386.27,A -85,B 0,C 180,E1 -8899.312,E2 -8899.312} C_VEL
LIN {X 0,Y 440.172,Z 394.182,A -85,B 0,C 180,E1 -8900.116,E2 -8900.116} C_VEL
LIN {X 0,Y 439.855,Z 399.863,A -85,B 0,C 180,E1 -8900.805,E2 -8900.805} C_VEL
LIN {X 0,Y 439.512,Z 406.199,A -85,B 0,C 180,E1 -8901.725,E2 -8901.725} C_VEL
LIN {X 0,Y 439.283,Z 411.806,A -85,B 0,C 180,E1 -8902.715,E2 -8902.715} C_VEL
LIN {X 0,Y 439.068,Z 415.853,A -85,B 0,C 180,E1 -8903.566,E2 -8903.566} C_VEL
LIN {X 0,Y 438.836,Z 419.513,A -85,B 0,C 180,E1 -8904.485,E2 -8904.485} C_VEL
LIN {X 0,Y 438.783,Z 422.492,A -85,B 0,C 180,E1 -8905.406,E2 -8905.406} C_VEL
LIN {X 0,Y 438.669,Z 424.803,A -85,B 0,C 180,E1 -8906.325,E2 -8906.325} C_VEL
LIN {X 0,Y 438.539,Z 426.566,A -85,B 0,C 180,E1 -8907.244,E2 -8907.244} C_VEL
LIN {X 0,Y 438.427,Z 427.84,A -85,B 0,C 180,E1 -8908.162,E2 -8908.162} C_VEL
LIN {X 0,Y 438.379,Z 428.644,A -85,B 0,C 180,E1 -8909.081,E2 -8909.081} C_VEL
LIN {X 0,Y 438.355,Z 428.951,A -85,B 0,C 180,E1 -8910,E2 -8910} C_VEL
LIN {X 0,Y 438.38,Z 428.677,A -85,B 0,C 180,E1 -8910.918,E2 -8910.918} C_VEL
LIN {X 0,Y 438.426,Z 427.939,A -85,B 0,C 180,E1 -8911.837,E2 -8911.837} C_VEL
LIN {X 0,Y 438.529,Z 426.733,A -85,B 0,C 180,E1 -8912.755,E2 -8912.755} C_VEL
LIN {X 0,Y 438.713,Z 423.899,A -85,B 0,C 180,E1 -8914.133,E2 -8914.133} C_VEL
LIN {X 0,Y 438.852,Z 421.321,A -85,B 0,C 180,E1 -8915.053,E2 -8915.053} C_VEL
LIN {X 0,Y 438.884,Z 418.145,A -85,B 0,C 180,E1 -8915.974,E2 -8915.974} C_VEL
LIN {X 0,Y 439.256,Z 413.935,A -85,B 0,C 180,E1 -8916.957,E2 -8916.957} C_VEL
LIN {X 0,Y 439.422,Z 408.189,A -85,B 0,C 180,E1 -8918.044,E2 -8918.044} C_VEL
LIN {X 0,Y 439.756,Z 402.246,A -85,B 0,C 180,E1 -8918.964,E2 -8918.964} C_VEL
LIN {X 0,Y 440.139,Z 395.008,A -85,B 0,C 180,E1 -8919.883,E2 -8919.883} C_VEL
LIN {X 0,Y 440.552,Z 387.268,A -85,B 0,C 180,E1 -8920.687,E2 -8920.687} C_VEL
LIN {X 0,Y 440.764,Z 379.111,A -85,B 0,C 180,E1 -8921.38,E2 -8921.38} C_VEL
LIN {X 0,Y 441.168,Z 370.58,A -85,B 0,C 180,E1 -8921.952,E2 -8921.952} C_VEL
LIN {X 0,Y 441.42,Z 359.307,A -85,B 0,C 180,E1 -8922.528,E2 -8922.528} C_VEL
LIN {X 0,Y 441.542,Z 348.1,A -85,B 0,C 180,E1 -8922.893,E2 -8922.893} C_VEL
LIN {X 0,Y 441.858,Z 325.792,A -85,B 0,C 180,E1 -8923.286,E2 -8923.286} C_VEL
LIN {X 0,Y 442.011,Z 282.77,A -85,B 0,C 180,E1 -8923.987,E2 -8923.987} C_VEL
LIN {X 0,Y 439.538,Z 269.776,A -85,B 0,C 180,E1 -8924.29,E2 -8924.29} C_VEL
LIN {X 0,Y 439.404,Z 261.097,A -85,B 0,C 180,E1 -8926.328,E2 -8926.328} C_VEL
LIN {X 0,Y 439.315,Z 260.58,A -85,B 0,C 180,E1 -8926.526,E2 -8926.526} C_VEL
LIN {X 0,Y 439.399,Z 260.568,A -85,B 0,C 180,E1 -8929.626,E2 -8929.626} C_VEL
LIN {X 0,Y 439.353,Z 260.57,A -85,B 0,C 180,E1 -8932.575,E2 -8932.575} C_VEL
LIN {X 0,Y 439.364,Z 260.568,A -85,B 0,C 180,E1 -8935.587,E2 -8935.587} C_VEL
LIN {X 0,Y 439.378,Z 260.568,A -85,B 0,C 180,E1 -8938.676,E2 -8938.676} C_VEL
LIN {X 0,Y 439.35,Z 260.57,A -85,B 0,C 180,E1 -8942.026,E2 -8942.026} C_VEL
LIN {X 0,Y 439.387,Z 260.565,A -85,B 0,C 180,E1 -8945.339,E2 -8945.339} C_VEL
LIN {X 0,Y 439.359,Z 260.571,A -85,B 0,C 180,E1 -8948.597,E2 -8948.597} C_VEL
LIN {X 0,Y 439.345,Z 260.571,A -85,B 0,C 180,E1 -8952.209,E2 -8952.209} C_VEL
LIN {X 0,Y 439.371,Z 260.568,A -85,B 0,C 180,E1 -8955.267,E2 -8955.267} C_VEL
LIN {X 0,Y 439.358,Z 260.569,A -85,B 0,C 180,E1 -8958.747,E2 -8958.747} C_VEL
LIN {X 0,Y 439.357,Z 260.569,A -85,B 0,C 180,E1 -8961.609,E2 -8961.609} C_VEL
LIN {X 0,Y 439.39,Z 260.565,A -85,B 0,C 180,E1 -8964.843,E2 -8964.843} C_VEL
LIN {X 0,Y 439.361,Z 260.57,A -85,B 0,C 180,E1 -8968.138,E2 -8968.138} C_VEL
LIN {X 0,Y 439.381,Z 260.566,A -85,B 0,C 180,E1 -8971.609,E2 -8971.609} C_VEL
LIN {X 0,Y 439.361,Z 260.568,A -85,B 0,C 180,E1 -8974.412,E2 -8974.412} C_VEL
LIN {X 0,Y 439.355,Z 260.569,A -85,B 0,C 180,E1 -8977.424,E2 -8977.424} C_VEL
LIN {X 0,Y 439.435,Z 260.561,A -85,B 0,C 180,E1 -8980.663,E2 -8980.663} C_VEL
LIN {X 0,Y 439.413,Z 260.562,A -85,B 0,C 180,E1 -8984.223,E2 -8984.223} C_VEL
LIN {X 0,Y 439.479,Z 260.554,A -85,B 0,C 180,E1 -8987.285,E2 -8987.285} C_VEL
LIN {X 0,Y 439.469,Z 260.556,A -85,B 0,C 180,E1 -8990.798,E2 -8990.798} C_VEL
LIN {X 0,Y 439.553,Z 260.544,A -85,B 0,C 180,E1 -8993.574,E2 -8993.574} C_VEL
LIN {X 0,Y 439.399,Z 260.564,A -85,B 0,C 180,E1 -8995.413,E2 -8995.413} C_VEL
LIN {X 0,Y 439.62,Z 260.538,A -85,B 0,C 180,E1 -8998.168,E2 -8998.168} C_VEL
LIN {X 0,Y 439.663,Z 260.532,A -85,B 0,C 180,E1 -9000,E2 -9000} C_VEL
LIN {X 0,Y 439.597,Z 260.539,A -85,B 0,C 180,E1 -9002.749,E2 -9002.749} C_VEL
LIN {X 0,Y 439.551,Z 260.545,A -85,B 0,C 180,E1 -9006.426,E2 -9006.426} C_VEL
LIN {X 0,Y 439.468,Z 260.554,A -85,B 0,C 180,E1 -9009.202,E2 -9009.202} C_VEL
LIN {X 0,Y 439.459,Z 260.556,A -85,B 0,C 180,E1 -9012.938,E2 -9012.938} C_VEL
LIN {X 0,Y 439.395,Z 260.564,A -85,B 0,C 180,E1 -9016.328,E2 -9016.328} C_VEL
LIN {X 0,Y 439.371,Z 260.569,A -85,B 0,C 180,E1 -9019.628,E2 -9019.628} C_VEL
LIN {X 0,Y 439.346,Z 260.569,A -85,B 0,C 180,E1 -9022.576,E2 -9022.576} C_VEL
LIN {X 0,Y 439.36,Z 260.572,A -85,B 0,C 180,E1 -9025.588,E2 -9025.588} C_VEL
LIN {X 0,Y 439.37,Z 260.566,A -85,B 0,C 180,E1 -9028.677,E2 -9028.677} C_VEL
LIN {X 0,Y 439.346,Z 260.569,A -85,B 0,C 180,E1 -9032.027,E2 -9032.027} C_VEL
LIN {X 0,Y 439.381,Z 260.57,A -85,B 0,C 180,E1 -9035.339,E2 -9035.339} C_VEL
LIN {X 0,Y 439.349,Z 260.568,A -85,B 0,C 180,E1 -9038.598,E2 -9038.598} C_VEL
LIN {X 0,Y 439.343,Z 260.568,A -85,B 0,C 180,E1 -9042.21,E2 -9042.21} C_VEL
LIN {X 0,Y 439.392,Z 260.566,A -85,B 0,C 180,E1 -9045.27,E2 -9045.27} C_VEL
LIN {X 0,Y 439.349,Z 260.574,A -85,B 0,C 180,E1 -9049.017,E2 -9049.017} C_VEL
LIN {X 0,Y 439.351,Z 260.567,A -85,B 0,C 180,E1 -9051.612,E2 -9051.612} C_VEL
LIN {X 0,Y 439.384,Z 260.569,A -85,B 0,C 180,E1 -9054.843,E2 -9054.843} C_VEL
LIN {X 0,Y 439.341,Z 260.569,A -85,B 0,C 180,E1 -9058.138,E2 -9058.138} C_VEL
LIN {X 0,Y 439.373,Z 260.567,A -85,B 0,C 180,E1 -9061.324,E2 -9061.324} C_VEL
LIN {X 0,Y 439.442,Z 260.734,A -85,B 0,C 180,E1 -9064.608,E2 -9064.608} C_VEL
LIN {X 0,Y 441.042,Z 269.673,A -85,B 0,C 180,E1 -9066.524,E2 -9066.524} C_VEL
LIN {X 0,Y 440.591,Z 281.812,A -85,B 0,C 180,E1 -9068.968,E2 -9068.968} C_VEL
LIN {X 0,Y 439.965,Z 296.315,A -85,B 0,C 180,E1 -9071.851,E2 -9071.851} C_VEL
LIN {X 0,Y 439.419,Z 311.962,A -85,B 0,C 180,E1 -9074.936,E2 -9074.936} C_VEL
LIN {X 0,Y 439.269,Z 316.232,A -85,B 0,C 180,E1 -9075.742,E2 -9075.742} C_VEL
LIN {X 0,Y 441.726,Z 337.347,A -85,B 0,C 180,E1 -9076.167,E2 -9076.167} C_VEL
LIN {X 0,Y 441.345,Z 393.688,A -85,B 0,C 180,E1 -9077.102,E2 -9077.102} C_VEL
LIN {X 0,Y 441.082,Z 403.205,A -85,B 0,C 180,E1 -9077.374,E2 -9077.374} C_VEL
LIN {X 0,Y 440.719,Z 413.267,A -85,B 0,C 180,E1 -9077.802,E2 -9077.802} C_VEL
LIN {X 0,Y 440.232,Z 424.705,A -85,B 0,C 180,E1 -9078.49,E2 -9078.49} C_VEL
LIN {X 0,Y 439.822,Z 433.317,A -85,B 0,C 180,E1 -9079.179,E2 -9079.179} C_VEL
LIN {X 0,Y 439.489,Z 441.428,A -85,B 0,C 180,E1 -9079.986,E2 -9079.986} C_VEL
LIN {X 0,Y 439.138,Z 448.128,A -85,B 0,C 180,E1 -9080.791,E2 -9080.791} C_VEL
LIN {X 0,Y 438.845,Z 454.494,A -85,B 0,C 180,E1 -9081.713,E2 -9081.713} C_VEL
LIN {X 0,Y 438.712,Z 459.792,A -85,B 0,C 180,E1 -9082.637,E2 -9082.637} C_VEL
LIN {X 0,Y 438.503,Z 464.206,A -85,B 0,C 180,E1 -9083.559,E2 -9083.559} C_VEL
LIN {X 0,Y 438.427,Z 467.886,A -85,B 0,C 180,E1 -9084.481,E2 -9084.481} C_VEL
LIN {X 0,Y 438.373,Z 470.906,A -85,B 0,C 180,E1 -9085.403,E2 -9085.403} C_VEL
LIN {X 0,Y 438.353,Z 473.249,A -85,B 0,C 180,E1 -9086.324,E2 -9086.324} C_VEL
LIN {X 0,Y 438.4,Z 475.015,A -85,B 0,C 180,E1 -9087.244,E2 -9087.244} C_VEL
LIN {X 0,Y 438.343,Z 476.275,A -85,B 0,C 180,E1 -9088.163,E2 -9088.163} C_VEL
LIN {X 0,Y 438.352,Z 477.061,A -85,B 0,C 180,E1 -9089.082,E2 -9089.082} C_VEL
LIN {X 0,Y 438.348,Z 477.358,A -85,B 0,C 180,E1 -9090,E2 -9090} C_VEL
LIN {X 0,Y 438.352,Z 477.059,A -85,B 0,C 180,E1 -9090.919,E2 -9090.919} C_VEL
LIN {X 0,Y 438.343,Z 476.27,A -85,B 0,C 180,E1 -9091.838,E2 -9091.838} C_VEL
LIN {X 0,Y 438.4,Z 475.007,A -85,B 0,C 180,E1 -9092.757,E2 -9092.757} C_VEL
LIN {X 0,Y 438.338,Z 472.073,A -85,B 0,C 180,E1 -9094.138,E2 -9094.138} C_VEL
LIN {X 0,Y 438.442,Z 469.408,A -85,B 0,C 180,E1 -9095.058,E2 -9095.058} C_VEL
LIN {X 0,Y 438.443,Z 465.627,A -85,B 0,C 180,E1 -9096.098,E2 -9096.098} C_VEL
LIN {X 0,Y 438.626,Z 460.945,A -85,B 0,C 180,E1 -9097.134,E2 -9097.134} C_VEL
LIN {X 0,Y 438.78,Z 455.891,A -85,B 0,C 180,E1 -9098.057,E2 -9098.057} C_VEL
LIN {X 0,Y 439.077,Z 449.813,A -85,B 0,C 180,E1 -9098.979,E2 -9098.979} C_VEL
LIN {X 0,Y 439.415,Z 442.418,A -85,B 0,C 180,E1 -9099.901,E2 -9099.901} C_VEL
LIN {X 0,Y 439.79,Z 434.506,A -85,B 0,C 180,E1 -9100.707,E2 -9100.707} C_VEL
LIN {X 0,Y 440.168,Z 426.151,A -85,B 0,C 180,E1 -9101.396,E2 -9101.396} C_VEL
LIN {X 0,Y 440.675,Z 415.491,A -85,B 0,C 180,E1 -9102.083,E2 -9102.083} C_VEL
LIN {X 0,Y 441.056,Z 403.898,A -85,B 0,C 180,E1 -9102.598,E2 -9102.598} C_VEL
LIN {X 0,Y 441.314,Z 394.205,A -85,B 0,C 180,E1 -9102.883,E2 -9102.883} C_VEL
LIN {X 0,Y 441.626,Z 360.45,A -85,B 0,C 180,E1 -9103.454,E2 -9103.454} C_VEL
LIN {X 0,Y 441.621,Z 337.028,A -85,B 0,C 180,E1 -9103.837,E2 -9103.837} C_VEL
LIN {X 0,Y 439.279,Z 315.925,A -85,B 0,C 180,E1 -9104.282,E2 -9104.282} C_VEL
LIN {X 0,Y 439.927,Z 297.491,A -85,B 0,C 180,E1 -9107.911,E2 -9107.911} C_VEL
LIN {X 0,Y 440.491,Z 284.202,A -85,B 0,C 180,E1 -9110.549,E2 -9110.549} C_VEL
LIN {X 0,Y 441.098,Z 270.86,A -85,B 0,C 180,E1 -9113.225,E2 -9113.225} C_VEL
LIN {X 0,Y 439.5,Z 261.004,A -85,B 0,C 180,E1 -9115.326,E2 -9115.326} C_VEL
LIN {X 0,Y 439.409,Z 260.565,A -85,B 0,C 180,E1 -9115.458,E2 -9115.458} C_VEL
LIN {X 0,Y 439.376,Z 260.565,A -85,B 0,C 180,E1 -9118.677,E2 -9118.677} C_VEL
LIN {X 0,Y 439.342,Z 260.568,A -85,B 0,C 180,E1 -9122.025,E2 -9122.025} C_VEL
LIN {X 0,Y 439.382,Z 260.567,A -85,B 0,C 180,E1 -9125.338,E2 -9125.338} C_VEL
LIN {X 0,Y 439.347,Z 260.569,A -85,B 0,C 180,E1 -9128.599,E2 -9128.599} C_VEL
LIN {X 0,Y 439.344,Z 260.568,A -85,B 0,C 180,E1 -9132.211,E2 -9132.211} C_VEL
LIN {X 0,Y 439.396,Z 260.564,A -85,B 0,C 180,E1 -9135.27,E2 -9135.27} C_VEL
LIN {X 0,Y 439.351,Z 260.571,A -85,B 0,C 180,E1 -9139.016,E2 -9139.016} C_VEL
LIN {X 0,Y 439.353,Z 260.567,A -85,B 0,C 180,E1 -9141.612,E2 -9141.612} C_VEL
LIN {X 0,Y 439.388,Z 260.567,A -85,B 0,C 180,E1 -9144.843,E2 -9144.843} C_VEL
LIN {X 0,Y 439.345,Z 260.57,A -85,B 0,C 180,E1 -9148.137,E2 -9148.137} C_VEL
LIN {X 0,Y 439.377,Z 260.565,A -85,B 0,C 180,E1 -9151.324,E2 -9151.324} C_VEL
LIN {X 0,Y 439.351,Z 260.573,A -85,B 0,C 180,E1 -9154.412,E2 -9154.412} C_VEL
LIN {X 0,Y 439.349,Z 260.569,A -85,B 0,C 180,E1 -9157.424,E2 -9157.424} C_VEL
LIN {X 0,Y 439.381,Z 260.566,A -85,B 0,C 180,E1 -9160.686,E2 -9160.686} C_VEL
LIN {X 0,Y 439.401,Z 260.566,A -85,B 0,C 180,E1 -9164.222,E2 -9164.222} C_VEL
LIN {X 0,Y 439.467,Z 260.555,A -85,B 0,C 180,E1 -9167.297,E2 -9167.297} C_VEL
LIN {X 0,Y 439.473,Z 260.554,A -85,B 0,C 180,E1 -9170.798,E2 -9170.798} C_VEL
LIN {X 0,Y 439.559,Z 260.544,A -85,B 0,C 180,E1 -9173.574,E2 -9173.574} C_VEL
LIN {X 0,Y 439.403,Z 260.563,A -85,B 0,C 180,E1 -9175.413,E2 -9175.413} C_VEL
LIN {X 0,Y 439.627,Z 260.536,A -85,B 0,C 180,E1 -9178.168,E2 -9178.168} C_VEL
LIN {X 0,Y 439.669,Z 260.531,A -85,B 0,C 180,E1 -9180,E2 -9180} C_VEL
LIN {X 0,Y 439.603,Z 260.539,A -85,B 0,C 180,E1 -9182.749,E2 -9182.749} C_VEL
LIN {X 0,Y 439.559,Z 260.544,A -85,B 0,C 180,E1 -9186.426,E2 -9186.426} C_VEL
LIN {X 0,Y 439.474,Z 260.555,A -85,B 0,C 180,E1 -9189.202,E2 -9189.202} C_VEL
LIN {X 0,Y 439.466,Z 260.555,A -85,B 0,C 180,E1 -9192.938,E2 -9192.938} C_VEL
LIN {X 0,Y 439.398,Z 260.565,A -85,B 0,C 180,E1 -9196.326,E2 -9196.326} C_VEL
LIN {X 0,Y 439.378,Z 260.566,A -85,B 0,C 180,E1 -9199.628,E2 -9199.628} C_VEL
LIN {X 0,Y 439.354,Z 260.569,A -85,B 0,C 180,E1 -9202.576,E2 -9202.576} C_VEL
LIN {X 0,Y 439.367,Z 260.568,A -85,B 0,C 180,E1 -9205.587,E2 -9205.587} C_VEL
LIN {X 0,Y 439.381,Z 260.566,A -85,B 0,C 180,E1 -9208.676,E2 -9208.676} C_VEL
LIN {X 0,Y 439.364,Z 260.57,A -85,B 0,C 180,E1 -9212.029,E2 -9212.029} C_VEL
LIN {X 0,Y 439.391,Z 260.565,A -85,B 0,C 180,E1 -9215.339,E2 -9215.339} C_VEL
LIN {X 0,Y 439.361,Z 260.569,A -85,B 0,C 180,E1 -9218.597,E2 -9218.597} C_VEL
LIN {X 0,Y 439.35,Z 260.57,A -85,B 0,C 180,E1 -9222.21,E2 -9222.21} C_VEL
LIN {X 0,Y 439.377,Z 260.567,A -85,B 0,C 180,E1 -9225.267,E2 -9225.267} C_VEL
LIN {X 0,Y 439.364,Z 260.568,A -85,B 0,C 180,E1 -9228.747,E2 -9228.747} C_VEL
LIN {X 0,Y 439.366,Z 260.57,A -85,B 0,C 180,E1 -9231.609,E2 -9231.609} C_VEL
LIN {X 0,Y 439.397,Z 260.564,A -85,B 0,C 180,E1 -9234.843,E2 -9234.843} C_VEL
LIN {X 0,Y 439.355,Z 260.569,A -85,B 0,C 180,E1 -9238.138,E2 -9238.138} C_VEL
LIN {X 0,Y 439.382,Z 260.568,A -85,B 0,C 180,E1 -9241.324,E2 -9241.324} C_VEL
LIN {X 0,Y 439.373,Z 260.567,A -85,B 0,C 180,E1 -9244.413,E2 -9244.413} C_VEL
LIN {X 0,Y 439.362,Z 260.569,A -85,B 0,C 180,E1 -9247.424,E2 -9247.424} C_VEL
LIN {X 0,Y 439.443,Z 260.565,A -85,B 0,C 180,E1 -9250.663,E2 -9250.663} C_VEL
LIN {X 0,Y 439.381,Z 260.746,A -85,B 0,C 180,E1 -9253.682,E2 -9253.682} C_VEL
LIN {X 0,Y 439.562,Z 268.18,A -85,B 0,C 180,E1 -9255.438,E2 -9255.438} C_VEL
LIN {X 0,Y 439.598,Z 269.991,A -85,B 0,C 180,E1 -9255.816,E2 -9255.816} C_VEL
LIN {X 0,Y 442.134,Z 283.349,A -85,B 0,C 180,E1 -9256.121,E2 -9256.121} C_VEL
LIN {X 0,Y 441.559,Z 345.979,A -85,B 0,C 180,E1 -9257.154,E2 -9257.154} C_VEL
LIN {X 0,Y 441.426,Z 355.064,A -85,B 0,C 180,E1 -9257.413,E2 -9257.413} C_VEL
LIN {X 0,Y 441.38,Z 359.502,A -85,B 0,C 180,E1 -9257.574,E2 -9257.574} C_VEL
LIN {X 0,Y 440.696,Z 365.084,A -85,B 0,C 180,E1 -9257.808,E2 -9257.808} C_VEL
LIN {X 0,Y 437.694,Z 373.946,A -85,B 0,C 180,E1 -9258.235,E2 -9258.235} C_VEL
LIN {X 0,Y 434.511,Z 382.42,A -85,B 0,C 180,E1 -9258.779,E2 -9258.779} C_VEL
LIN {X 0,Y 433.554,Z 387.276,A -85,B 0,C 180,E1 -9259.196,E2 -9259.196} C_VEL
LIN {X 0,Y 433.211,Z 394.576,A -85,B 0,C 180,E1 -9259.956,E2 -9259.956} C_VEL
LIN {X 0,Y 432.873,Z 400.257,A -85,B 0,C 180,E1 -9260.656,E2 -9260.656} C_VEL
LIN {X 0,Y 432.512,Z 406.592,A -85,B 0,C 180,E1 -9261.59,E2 -9261.59} C_VEL
LIN {X 0,Y 432.229,Z 412.632,A -85,B 0,C 180,E1 -9262.683,E2 -9262.683} C_VEL
LIN {X 0,Y 432.051,Z 416.244,A -85,B 0,C 180,E1 -9263.461,E2 -9263.461} C_VEL
LIN {X 0,Y 431.775,Z 419.906,A -85,B 0,C 180,E1 -9264.395,E2 -9264.395} C_VEL
LIN {X 0,Y 431.715,Z 422.884,A -85,B 0,C 180,E1 -9265.331,E2 -9265.331} C_VEL
LIN {X 0,Y 431.612,Z 425.194,A -85,B 0,C 180,E1 -9266.265,E2 -9266.265} C_VEL
LIN {X 0,Y 431.468,Z 426.958,A -85,B 0,C 180,E1 -9267.199,E2 -9267.199} C_VEL
LIN {X 0,Y 431.346,Z 428.231,A -85,B 0,C 180,E1 -9268.132,E2 -9268.132} C_VEL
LIN {X 0,Y 431.304,Z 429.035,A -85,B 0,C 180,E1 -9269.066,E2 -9269.066} C_VEL
LIN {X 0,Y 431.294,Z 429.34,A -85,B 0,C 180,E1 -9270,E2 -9270} C_VEL
LIN {X 0,Y 431.304,Z 429.067,A -85,B 0,C 180,E1 -9270.933,E2 -9270.933} C_VEL
LIN {X 0,Y 431.345,Z 428.329,A -85,B 0,C 180,E1 -9271.867,E2 -9271.867} C_VEL
LIN {X 0,Y 431.458,Z 427.123,A -85,B 0,C 180,E1 -9272.8,E2 -9272.8} C_VEL
LIN {X 0,Y 431.661,Z 424.288,A -85,B 0,C 180,E1 -9274.201,E2 -9274.201} C_VEL
LIN {X 0,Y 431.78,Z 421.712,A -85,B 0,C 180,E1 -9275.136,E2 -9275.136} C_VEL
LIN {X 0,Y 431.852,Z 418.534,A -85,B 0,C 180,E1 -9276.072,E2 -9276.072} C_VEL
LIN {X 0,Y 432.254,Z 412.974,A -85,B 0,C 180,E1 -9277.343,E2 -9277.343} C_VEL
LIN {X 0,Y 432.482,Z 407.168,A -85,B 0,C 180,E1 -9278.409,E2 -9278.409} C_VEL
LIN {X 0,Y 432.864,Z 400.94,A -85,B 0,C 180,E1 -9279.343,E2 -9279.343} C_VEL
LIN {X 0,Y 433.326,Z 393.362,A -85,B 0,C 180,E1 -9280.276,E2 -9280.276} C_VEL
LIN {X 0,Y 433.731,Z 383.933,A -85,B 0,C 180,E1 -9281.212,E2 -9281.212} C_VEL
LIN {X 0,Y 434.087,Z 374.698,A -85,B 0,C 180,E1 -9281.912,E2 -9281.912} C_VEL
LIN {X 0,Y 434.407,Z 364.572,A -85,B 0,C 180,E1 -9282.496,E2 -9282.496} C_VEL
LIN {X 0,Y 434.534,Z 355.66,A -85,B 0,C 180,E1 -9282.878,E2 -9282.878} C_VEL
LIN {X 0,Y 434.708,Z 346.144,A -85,B 0,C 180,E1 -9283.153,E2 -9283.153} C_VEL
LIN {X 0,Y 435.122,Z 283.414,A -85,B 0,C 180,E1 -9284.208,E2 -9284.208} C_VEL
LIN {X 0,Y 432.577,Z 270.148,A -85,B 0,C 180,E1 -9284.525,E2 -9284.525} C_VEL
LIN {X 0,Y 432.373,Z 262.021,A -85,B 0,C 180,E1 -9286.46,E2 -9286.46} C_VEL
LIN {X 0,Y 432.289,Z 261.455,A -85,B 0,C 180,E1 -9286.659,E2 -9286.659} C_VEL
LIN {X 0,Y 432.386,Z 261.443,A -85,B 0,C 180,E1 -9289.484,E2 -9289.484} C_VEL
LIN {X 0,Y 432.302,Z 261.451,A -85,B 0,C 180,E1 -9292.965,E2 -9292.965} C_VEL
LIN {X 0,Y 432.316,Z 261.447,A -85,B 0,C 180,E1 -9296.035,E2 -9296.035} C_VEL
LIN {X 0,Y 432.319,Z 261.446,A -85,B 0,C 180,E1 -9299.189,E2 -9299.189} C_VEL
LIN {X 0,Y 432.313,Z 261.447,A -85,B 0,C 180,E1 -9302.443,E2 -9302.443} C_VEL
LIN {X 0,Y 432.333,Z 261.445,A -85,B 0,C 180,E1 -9305.817,E2 -9305.817} C_VEL
LIN {X 0,Y 432.299,Z 261.448,A -85,B 0,C 180,E1 -9309.347,E2 -9309.347} C_VEL
LIN {X 0,Y 432.3,Z 261.449,A -85,B 0,C 180,E1 -9311.8,E2 -9311.8} C_VEL
LIN {X 0,Y 432.328,Z 261.447,A -85,B 0,C 180,E1 -9314.347,E2 -9314.347} C_VEL
LIN {X 0,Y 432.298,Z 261.448,A -85,B 0,C 180,E1 -9317.018,E2 -9317.018} C_VEL
LIN {X 0,Y 432.284,Z 261.45,A -85,B 0,C 180,E1 -9319.827,E2 -9319.827} C_VEL
LIN {X 0,Y 432.298,Z 261.449,A -85,B 0,C 180,E1 -9323.021,E2 -9323.021} C_VEL
LIN {X 0,Y 432.328,Z 261.446,A -85,B 0,C 180,E1 -9326.001,E2 -9326.001} C_VEL
LIN {X 0,Y 432.335,Z 261.444,A -85,B 0,C 180,E1 -9329.491,E2 -9329.491} C_VEL
LIN {X 0,Y 432.314,Z 261.448,A -85,B 0,C 180,E1 -9331.872,E2 -9331.872} C_VEL
LIN {X 0,Y 432.318,Z 261.448,A -85,B 0,C 180,E1 -9334.997,E2 -9334.997} C_VEL
LIN {X 0,Y 432.35,Z 261.442,A -85,B 0,C 180,E1 -9338.045,E2 -9338.045} C_VEL
LIN {X 0,Y 432.376,Z 261.44,A -85,B 0,C 180,E1 -9341.029,E2 -9341.029} C_VEL
LIN {X 0,Y 432.383,Z 261.437,A -85,B 0,C 180,E1 -9343.959,E2 -9343.959} C_VEL
LIN {X 0,Y 432.448,Z 261.429,A -85,B 0,C 180,E1 -9347.803,E2 -9347.803} C_VEL
LIN {X 0,Y 432.441,Z 261.43,A -85,B 0,C 180,E1 -9351.589,E2 -9351.589} C_VEL
LIN {X 0,Y 432.546,Z 261.42,A -85,B 0,C 180,E1 -9354.405,E2 -9354.405} C_VEL
LIN {X 0,Y 432.589,Z 261.413,A -85,B 0,C 180,E1 -9358.138,E2 -9358.138} C_VEL
LIN {X 0,Y 432.614,Z 261.409,A -85,B 0,C 180,E1 -9360,E2 -9360} C_VEL
LIN {X 0,Y 432.55,Z 261.417,A -85,B 0,C 180,E1 -9362.794,E2 -9362.794} C_VEL
LIN {X 0,Y 432.508,Z 261.422,A -85,B 0,C 180,E1 -9366.531,E2 -9366.531} C_VEL
LIN {X 0,Y 432.414,Z 261.433,A -85,B 0,C 180,E1 -9369.354,E2 -9369.354} C_VEL
LIN {X 0,Y 432.425,Z 261.432,A -85,B 0,C 180,E1 -9372.803,E2 -9372.803} C_VEL
LIN {X 0,Y 432.354,Z 261.441,A -85,B 0,C 180,E1 -9376.455,E2 -9376.455} C_VEL
LIN {X 0,Y 432.307,Z 261.449,A -85,B 0,C 180,E1 -9379.962,E2 -9379.962} C_VEL
LIN {X 0,Y 432.297,Z 261.447,A -85,B 0,C 180,E1 -9382.965,E2 -9382.965} C_VEL
LIN {X 0,Y 432.311,Z 261.446,A -85,B 0,C 180,E1 -9386.036,E2 -9386.036} C_VEL
LIN {X 0,Y 432.309,Z 261.447,A -85,B 0,C 180,E1 -9389.19,E2 -9389.19} C_VEL
LIN {X 0,Y 432.31,Z 261.445,A -85,B 0,C 180,E1 -9392.444,E2 -9392.444} C_VEL
LIN {X 0,Y 432.327,Z 261.444,A -85,B 0,C 180,E1 -9395.819,E2 -9395.819} C_VEL
LIN {X 0,Y 432.294,Z 261.451,A -85,B 0,C 180,E1 -9399.349,E2 -9399.349} C_VEL
LIN {X 0,Y 432.298,Z 261.447,A -85,B 0,C 180,E1 -9401.801,E2 -9401.801} C_VEL
LIN {X 0,Y 432.329,Z 261.442,A -85,B 0,C 180,E1 -9404.348,E2 -9404.348} C_VEL
LIN {X 0,Y 432.296,Z 261.452,A -85,B 0,C 180,E1 -9407.019,E2 -9407.019} C_VEL
LIN {X 0,Y 432.284,Z 261.448,A -85,B 0,C 180,E1 -9409.828,E2 -9409.828} C_VEL
LIN {X 0,Y 432.291,Z 261.451,A -85,B 0,C 180,E1 -9413.021,E2 -9413.021} C_VEL
LIN {X 0,Y 432.326,Z 261.442,A -85,B 0,C 180,E1 -9416.003,E2 -9416.003} C_VEL
LIN {X 0,Y 432.327,Z 261.442,A -85,B 0,C 180,E1 -9419.494,E2 -9419.494} C_VEL
LIN {X 0,Y 432.308,Z 261.447,A -85,B 0,C 180,E1 -9421.872,E2 -9421.872} C_VEL
LIN {X 0,Y 432.391,Z 261.548,A -85,B 0,C 180,E1 -9424.423,E2 -9424.423} C_VEL
LIN {X 0,Y 434.132,Z 271.713,A -85,B 0,C 180,E1 -9426.634,E2 -9426.634} C_VEL
LIN {X 0,Y 433.371,Z 287.467,A -85,B 0,C 180,E1 -9429.842,E2 -9429.842} C_VEL
LIN {X 0,Y 432.707,Z 303.151,A -85,B 0,C 180,E1 -9433.002,E2 -9433.002} C_VEL
LIN {X 0,Y 432.251,Z 315.85,A -85,B 0,C 180,E1 -9435.506,E2 -9435.506} C_VEL
LIN {X 0,Y 434.849,Z 338.569,A -85,B 0,C 180,E1 -9435.971,E2 -9435.971} C_VEL
LIN {X 0,Y 434.446,Z 392.632,A -85,B 0,C 180,E1 -9436.878,E2 -9436.878} C_VEL
LIN {X 0,Y 434.211,Z 401.99,A -85,B 0,C 180,E1 -9437.142,E2 -9437.142} C_VEL
LIN {X 0,Y 433.813,Z 411.668,A -85,B 0,C 180,E1 -9437.546,E2 -9437.546} C_VEL
LIN {X 0,Y 433.445,Z 420.852,A -85,B 0,C 180,E1 -9438.07,E2 -9438.07} C_VEL
LIN {X 0,Y 432.886,Z 431.689,A -85,B 0,C 180,E1 -9438.885,E2 -9438.885} C_VEL
LIN {X 0,Y 432.474,Z 441.037,A -85,B 0,C 180,E1 -9439.821,E2 -9439.821} C_VEL
LIN {X 0,Y 432.106,Z 447.737,A -85,B 0,C 180,E1 -9440.64,E2 -9440.64} C_VEL
LIN {X 0,Y 431.801,Z 454.103,A -85,B 0,C 180,E1 -9441.577,E2 -9441.577} C_VEL
LIN {X 0,Y 431.637,Z 459.4,A -85,B 0,C 180,E1 -9442.516,E2 -9442.516} C_VEL
LIN {X 0,Y 431.405,Z 464.373,A -85,B 0,C 180,E1 -9443.589,E2 -9443.589} C_VEL
LIN {X 0,Y 431.348,Z 469.03,A -85,B 0,C 180,E1 -9444.859,E2 -9444.859} C_VEL
LIN {X 0,Y 431.253,Z 472.857,A -85,B 0,C 180,E1 -9446.263,E2 -9446.263} C_VEL
LIN {X 0,Y 431.326,Z 474.625,A -85,B 0,C 180,E1 -9447.199,E2 -9447.199} C_VEL
LIN {X 0,Y 431.264,Z 475.884,A -85,B 0,C 180,E1 -9448.133,E2 -9448.133} C_VEL
LIN {X 0,Y 431.262,Z 476.67,A -85,B 0,C 180,E1 -9449.067,E2 -9449.067} C_VEL
LIN {X 0,Y 431.287,Z 476.968,A -85,B 0,C 180,E1 -9450,E2 -9450} C_VEL
LIN {X 0,Y 431.262,Z 476.668,A -85,B 0,C 180,E1 -9450.934,E2 -9450.934} C_VEL
LIN {X 0,Y 431.264,Z 475.879,A -85,B 0,C 180,E1 -9451.868,E2 -9451.868} C_VEL
LIN {X 0,Y 431.327,Z 474.615,A -85,B 0,C 180,E1 -9452.802,E2 -9452.802} C_VEL
LIN {X 0,Y 431.254,Z 471.68,A -85,B 0,C 180,E1 -9454.206,E2 -9454.206} C_VEL
LIN {X 0,Y 431.348,Z 469.013,A -85,B 0,C 180,E1 -9455.142,E2 -9455.142} C_VEL
LIN {X 0,Y 431.438,Z 463.792,A -85,B 0,C 180,E1 -9456.548,E2 -9456.548} C_VEL
LIN {X 0,Y 431.685,Z 456.92,A -85,B 0,C 180,E1 -9457.955,E2 -9457.955} C_VEL
LIN {X 0,Y 432.03,Z 449.416,A -85,B 0,C 180,E1 -9459.126,E2 -9459.126} C_VEL
LIN {X 0,Y 432.413,Z 442.023,A -85,B 0,C 180,E1 -9460.063,E2 -9460.063} C_VEL
LIN {X 0,Y 432.783,Z 434.109,A -85,B 0,C 180,E1 -9460.882,E2 -9460.882} C_VEL
LIN {X 0,Y 433.197,Z 425.754,A -85,B 0,C 180,E1 -9461.582,E2 -9461.582} C_VEL
LIN {X 0,Y 433.692,Z 415.091,A -85,B 0,C 180,E1 -9462.281,E2 -9462.281} C_VEL
LIN {X 0,Y 434.135,Z 403.498,A -85,B 0,C 180,E1 -9462.802,E2 -9462.802} C_VEL
LIN {X 0,Y 434.405,Z 393.8,A -85,B 0,C 180,E1 -9463.091,E2 -9463.091} C_VEL
LIN {X 0,Y 434.75,Z 358.993,A -85,B 0,C 180,E1 -9463.688,E2 -9463.688} C_VEL
LIN {X 0,Y 434.697,Z 336.905,A -85,B 0,C 180,E1 -9464.057,E2 -9464.057} C_VEL
LIN {X 0,Y 432.223,Z 315.528,A -85,B 0,C 180,E1 -9464.52,E2 -9464.52} C_VEL
LIN {X 0,Y 432.902,Z 298.299,A -85,B 0,C 180,E1 -9467.967,E2 -9467.967} C_VEL
LIN {X 0,Y 433.498,Z 285.015,A -85,B 0,C 180,E1 -9470.648,E2 -9470.648} C_VEL
LIN {X 0,Y 434.114,Z 271.676,A -85,B 0,C 180,E1 -9473.369,E2 -9473.369} C_VEL
LIN {X 0,Y 432.377,Z 261.441,A -85,B 0,C 180,E1 -9475.612,E2 -9475.612} C_VEL
LIN {X 0,Y 432.314,Z 261.449,A -85,B 0,C 180,E1 -9479.19,E2 -9479.19} C_VEL
LIN {X 0,Y 432.304,Z 261.445,A -85,B 0,C 180,E1 -9482.445,E2 -9482.445} C_VEL
LIN {X 0,Y 432.33,Z 261.442,A -85,B 0,C 180,E1 -9485.819,E2 -9485.819} C_VEL
LIN {X 0,Y 432.311,Z 261.446,A -85,B 0,C 180,E1 -9488.71,E2 -9488.71} C_VEL
LIN {X 0,Y 432.3,Z 261.445,A -85,B 0,C 180,E1 -9491.801,E2 -9491.801} C_VEL
LIN {X 0,Y 432.334,Z 261.442,A -85,B 0,C 180,E1 -9494.348,E2 -9494.348} C_VEL
LIN {X 0,Y 432.3,Z 261.45,A -85,B 0,C 180,E1 -9497.019,E2 -9497.019} C_VEL
LIN {X 0,Y 432.288,Z 261.448,A -85,B 0,C 180,E1 -9499.828,E2 -9499.828} C_VEL
LIN {X 0,Y 432.295,Z 261.449,A -85,B 0,C 180,E1 -9503.021,E2 -9503.021} C_VEL
LIN {X 0,Y 432.33,Z 261.443,A -85,B 0,C 180,E1 -9506.003,E2 -9506.003} C_VEL
LIN {X 0,Y 432.331,Z 261.442,A -85,B 0,C 180,E1 -9509.494,E2 -9509.494} C_VEL
LIN {X 0,Y 432.312,Z 261.446,A -85,B 0,C 180,E1 -9511.872,E2 -9511.872} C_VEL
LIN {X 0,Y 432.312,Z 261.445,A -85,B 0,C 180,E1 -9514.996,E2 -9514.996} C_VEL
LIN {X 0,Y 432.348,Z 261.443,A -85,B 0,C 180,E1 -9518.045,E2 -9518.045} C_VEL
LIN {X 0,Y 432.338,Z 261.442,A -85,B 0,C 180,E1 -9521.027,E2 -9521.027} C_VEL
LIN {X 0,Y 432.356,Z 261.442,A -85,B 0,C 180,E1 -9523.958,E2 -9523.958} C_VEL
LIN {X 0,Y 432.448,Z 261.431,A -85,B 0,C 180,E1 -9527.803,E2 -9527.803} C_VEL
LIN {X 0,Y 432.447,Z 261.43,A -85,B 0,C 180,E1 -9531.59,E2 -9531.59} C_VEL
LIN {X 0,Y 432.551,Z 261.416,A -85,B 0,C 180,E1 -9534.406,E2 -9534.406} C_VEL
LIN {X 0,Y 432.596,Z 261.411,A -85,B 0,C 180,E1 -9538.138,E2 -9538.138} C_VEL
LIN {X 0,Y 432.621,Z 261.409,A -85,B 0,C 180,E1 -9540,E2 -9540} C_VEL
LIN {X 0,Y 432.557,Z 261.417,A -85,B 0,C 180,E1 -9542.794,E2 -9542.794} C_VEL
LIN {X 0,Y 432.516,Z 261.421,A -85,B 0,C 180,E1 -9546.531,E2 -9546.531} C_VEL
LIN {X 0,Y 432.42,Z 261.435,A -85,B 0,C 180,E1 -9549.354,E2 -9549.354} C_VEL
LIN {X 0,Y 432.432,Z 261.432,A -85,B 0,C 180,E1 -9552.803,E2 -9552.803} C_VEL
LIN {X 0,Y 432.358,Z 261.442,A -85,B 0,C 180,E1 -9556.453,E2 -9556.453} C_VEL
LIN {X 0,Y 432.314,Z 261.446,A -85,B 0,C 180,E1 -9559.962,E2 -9559.962} C_VEL
LIN {X 0,Y 432.304,Z 261.449,A -85,B 0,C 180,E1 -9562.965,E2 -9562.965} C_VEL
LIN {X 0,Y 432.319,Z 261.446,A -85,B 0,C 180,E1 -9566.036,E2 -9566.036} C_VEL
LIN {X 0,Y 432.322,Z 261.446,A -85,B 0,C 180,E1 -9569.189,E2 -9569.189} C_VEL
LIN {X 0,Y 432.322,Z 261.446,A -85,B 0,C 180,E1 -9572.443,E2 -9572.443} C_VEL
LIN {X 0,Y 432.337,Z 261.445,A -85,B 0,C 180,E1 -9575.818,E2 -9575.818} C_VEL
LIN {X 0,Y 432.303,Z 261.447,A -85,B 0,C 180,E1 -9579.348,E2 -9579.348} C_VEL
LIN {X 0,Y 432.304,Z 261.449,A -85,B 0,C 180,E1 -9581.801,E2 -9581.801} C_VEL
LIN {X 0,Y 432.333,Z 261.444,A -85,B 0,C 180,E1 -9584.348,E2 -9584.348} C_VEL
LIN {X 0,Y 432.304,Z 261.447,A -85,B 0,C 180,E1 -9587.018,E2 -9587.018} C_VEL
LIN {X 0,Y 432.291,Z 261.45,A -85,B 0,C 180,E1 -9589.828,E2 -9589.828} C_VEL
LIN {X 0,Y 432.306,Z 261.447,A -85,B 0,C 180,E1 -9593.022,E2 -9593.022} C_VEL
LIN {X 0,Y 432.334,Z 261.444,A -85,B 0,C 180,E1 -9596.002,E2 -9596.002} C_VEL
LIN {X 0,Y 432.339,Z 261.445,A -85,B 0,C 180,E1 -9599.492,E2 -9599.492} C_VEL
LIN {X 0,Y 432.321,Z 261.446,A -85,B 0,C 180,E1 -9601.872,E2 -9601.872} C_VEL
LIN {X 0,Y 432.367,Z 261.44,A -85,B 0,C 180,E1 -9605.542,E2 -9605.542} C_VEL
LIN {X 0,Y 432.351,Z 261.444,A -85,B 0,C 180,E1 -9609.046,E2 -9609.046} C_VEL
LIN {X 0,Y 432.335,Z 261.444,A -85,B 0,C 180,E1 -9612.009,E2 -9612.009} C_VEL
LIN {X 0,Y 432.36,Z 261.647,A -85,B 0,C 180,E1 -9613.546,E2 -9613.546} C_VEL
LIN {X 0,Y 432.574,Z 268.549,A -85,B 0,C 180,E1 -9615.197,E2 -9615.197} C_VEL
LIN {X 0,Y 432.625,Z 270.416,A -85,B 0,C 180,E1 -9615.583,E2 -9615.583} C_VEL
LIN {X 0,Y 435.277,Z 284.317,A -85,B 0,C 180,E1 -9615.907,E2 -9615.907} C_VEL
LIN {X 0,Y 434.669,Z 346.389,A -85,B 0,C 180,E1 -9616.946,E2 -9616.946} C_VEL
LIN {X 0,Y 434.521,Z 355.467,A -85,B 0,C 180,E1 -9617.209,E2 -9617.209} C_VEL
LIN {X 0,Y 434.331,Z 365.038,A -85,B 0,C 180,E1 -9617.619,E2 -9617.619} C_VEL
LIN {X 0,Y 434.058,Z 375.054,A -85,B 0,C 180,E1 -9618.204,E2 -9618.204} C_VEL
LIN {X 0,Y 433.663,Z 385.441,A -85,B 0,C 180,E1 -9619.022,E2 -9619.022} C_VEL
LIN {X 0,Y 433.554,Z 387.276,A -85,B 0,C 180,E1 -9619.196,E2 -9619.196} C_VEL
LIN {X 0,Y 432.586,Z 392.151,A -85,B 0,C 180,E1 -9619.654,E2 -9619.654} C_VEL
LIN {X 0,Y 429.309,Z 399.476,A -85,B 0,C 180,E1 -9620.439,E2 -9620.439} C_VEL
LIN {X 0,Y 426.173,Z 406.13,A -85,B 0,C 180,E1 -9621.32,E2 -9621.32} C_VEL
LIN {X 0,Y 425.401,Z 409.74,A -85,B 0,C 180,E1 -9621.917,E2 -9621.917} C_VEL
LIN {X 0,Y 425.177,Z 414.938,A -85,B 0,C 180,E1 -9622.954,E2 -9622.954} C_VEL
LIN {X 0,Y 424.721,Z 420.299,A -85,B 0,C 180,E1 -9624.302,E2 -9624.302} C_VEL
LIN {X 0,Y 424.648,Z 423.277,A -85,B 0,C 180,E1 -9625.253,E2 -9625.253} C_VEL
LIN {X 0,Y 424.557,Z 425.586,A -85,B 0,C 180,E1 -9626.203,E2 -9626.203} C_VEL
LIN {X 0,Y 424.4,Z 427.349,A -85,B 0,C 180,E1 -9627.152,E2 -9627.152} C_VEL
LIN {X 0,Y 424.267,Z 428.623,A -85,B 0,C 180,E1 -9628.101,E2 -9628.101} C_VEL
LIN {X 0,Y 424.217,Z 429.426,A -85,B 0,C 180,E1 -9629.05,E2 -9629.05} C_VEL
LIN {X 0,Y 424.204,Z 429.732,A -85,B 0,C 180,E1 -9630,E2 -9630} C_VEL
LIN {X 0,Y 424.217,Z 429.458,A -85,B 0,C 180,E1 -9630.949,E2 -9630.949} C_VEL
LIN {X 0,Y 424.266,Z 428.72,A -85,B 0,C 180,E1 -9631.898,E2 -9631.898} C_VEL
LIN {X 0,Y 424.391,Z 427.513,A -85,B 0,C 180,E1 -9632.847,E2 -9632.847} C_VEL
LIN {X 0,Y 424.608,Z 424.677,A -85,B 0,C 180,E1 -9634.271,E2 -9634.271} C_VEL
LIN {X 0,Y 424.714,Z 422.102,A -85,B 0,C 180,E1 -9635.221,E2 -9635.221} C_VEL
LIN {X 0,Y 424.982,Z 417.024,A -85,B 0,C 180,E1 -9636.647,E2 -9636.647} C_VEL
LIN {X 0,Y 425.296,Z 411.558,A -85,B 0,C 180,E1 -9637.835,E2 -9637.835} C_VEL
LIN {X 0,Y 425.68,Z 404.691,A -85,B 0,C 180,E1 -9639.023,E2 -9639.023} C_VEL
LIN {X 0,Y 426.149,Z 396.796,A -85,B 0,C 180,E1 -9640.091,E2 -9640.091} C_VEL
LIN {X 0,Y 426.543,Z 389.266,A -85,B 0,C 180,E1 -9640.922,E2 -9640.922} C_VEL
LIN {X 0,Y 426.86,Z 381.373,A -85,B 0,C 180,E1 -9641.635,E2 -9641.635} C_VEL
LIN {X 0,Y 427.28,Z 373.213,A -85,B 0,C 180,E1 -9642.226,E2 -9642.226} C_VEL
LIN {X 0,Y 427.51,Z 364.954,A -85,B 0,C 180,E1 -9642.701,E2 -9642.701} C_VEL
LIN {X 0,Y 427.637,Z 356.038,A -85,B 0,C 180,E1 -9643.09,E2 -9643.09} C_VEL
LIN {X 0,Y 427.789,Z 346.619,A -85,B 0,C 180,E1 -9643.367,E2 -9643.367} C_VEL
LIN {X 0,Y 428.283,Z 284.419,A -85,B 0,C 180,E1 -9644.429,E2 -9644.429} C_VEL
LIN {X 0,Y 425.582,Z 270.52,A -85,B 0,C 180,E1 -9644.769,E2 -9644.769} C_VEL
LIN {X 0,Y 425.475,Z 264.124,A -85,B 0,C 180,E1 -9646.308,E2 -9646.308} C_VEL
LIN {X 0,Y 425.25,Z 262.332,A -85,B 0,C 180,E1 -9646.757,E2 -9646.757} C_VEL
LIN {X 0,Y 425.327,Z 262.321,A -85,B 0,C 180,E1 -9649.634,E2 -9649.634} C_VEL
LIN {X 0,Y 425.284,Z 262.322,A -85,B 0,C 180,E1 -9652.338,E2 -9652.338} C_VEL
LIN {X 0,Y 425.257,Z 262.325,A -85,B 0,C 180,E1 -9655.447,E2 -9655.447} C_VEL
LIN {X 0,Y 425.297,Z 262.322,A -85,B 0,C 180,E1 -9658.858,E2 -9658.858} C_VEL
LIN {X 0,Y 425.251,Z 262.327,A -85,B 0,C 180,E1 -9661.927,E2 -9661.927} C_VEL
LIN {X 0,Y 425.292,Z 262.32,A -85,B 0,C 180,E1 -9665.336,E2 -9665.336} C_VEL
LIN {X 0,Y 425.277,Z 262.323,A -85,B 0,C 180,E1 -9668.9,E2 -9668.9} C_VEL
LIN {X 0,Y 425.253,Z 262.326,A -85,B 0,C 180,E1 -9672.655,E2 -9672.655} C_VEL
LIN {X 0,Y 425.28,Z 262.323,A -85,B 0,C 180,E1 -9675.283,E2 -9675.283} C_VEL
LIN {X 0,Y 425.243,Z 262.327,A -85,B 0,C 180,E1 -9678.618,E2 -9678.618} C_VEL
LIN {X 0,Y 425.275,Z 262.323,A -85,B 0,C 180,E1 -9681.099,E2 -9681.099} C_VEL
LIN {X 0,Y 425.29,Z 262.321,A -85,B 0,C 180,E1 -9684.663,E2 -9684.663} C_VEL
LIN {X 0,Y 425.256,Z 262.327,A -85,B 0,C 180,E1 -9688.072,E2 -9688.072} C_VEL
LIN {X 0,Y 425.29,Z 262.322,A -85,B 0,C 180,E1 -9691.365,E2 -9691.365} C_VEL
LIN {X 0,Y 425.254,Z 262.325,A -85,B 0,C 180,E1 -9694.552,E2 -9694.552} C_VEL
LIN {X 0,Y 425.286,Z 262.323,A -85,B 0,C 180,E1 -9697.73,E2 -9697.73} C_VEL
LIN {X 0,Y 425.355,Z 262.314,A -85,B 0,C 180,E1 -9700.704,E2 -9700.704} C_VEL
LIN {X 0,Y 425.317,Z 262.318,A -85,B 0,C 180,E1 -9703.685,E2 -9703.685} C_VEL
LIN {X 0,Y 425.388,Z 262.31,A -85,B 0,C 180,E1 -9707.097,E2 -9707.097} C_VEL
LIN {X 0,Y 425.375,Z 262.313,A -85,B 0,C 180,E1 -9710.49,E2 -9710.49} C_VEL
LIN {X 0,Y 425.471,Z 262.299,A -85,B 0,C 180,E1 -9713.36,E2 -9713.36} C_VEL
LIN {X 0,Y 425.338,Z 262.316,A -85,B 0,C 180,E1 -9715.261,E2 -9715.261} C_VEL
LIN {X 0,Y 425.558,Z 262.288,A -85,B 0,C 180,E1 -9718.107,E2 -9718.107} C_VEL
LIN {X 0,Y 425.566,Z 262.287,A -85,B 0,C 180,E1 -9720,E2 -9720} C_VEL
LIN {X 0,Y 425.506,Z 262.294,A -85,B 0,C 180,E1 -9722.84,E2 -9722.84} C_VEL
LIN {X 0,Y 425.469,Z 262.299,A -85,B 0,C 180,E1 -9726.64,E2 -9726.64} C_VEL
LIN {X 0,Y 425.375,Z 262.31,A -85,B 0,C 180,E1 -9729.51,E2 -9729.51} C_VEL
LIN {X 0,Y 425.387,Z 262.308,A -85,B 0,C 180,E1 -9732.903,E2 -9732.903} C_VEL
LIN {X 0,Y 425.311,Z 262.318,A -85,B 0,C 180,E1 -9736.584,E2 -9736.584} C_VEL
LIN {X 0,Y 425.29,Z 262.323,A -85,B 0,C 180,E1 -9739.623,E2 -9739.623} C_VEL
LIN {X 0,Y 425.279,Z 262.322,A -85,B 0,C 180,E1 -9742.339,E2 -9742.339} C_VEL
LIN {X 0,Y 425.253,Z 262.327,A -85,B 0,C 180,E1 -9745.448,E2 -9745.448} C_VEL
LIN {X 0,Y 425.289,Z 262.32,A -85,B 0,C 180,E1 -9748.857,E2 -9748.857} C_VEL
LIN {X 0,Y 425.247,Z 262.326,A -85,B 0,C 180,E1 -9751.928,E2 -9751.928} C_VEL
LIN {X 0,Y 425.287,Z 262.325,A -85,B 0,C 180,E1 -9755.337,E2 -9755.337} C_VEL
LIN {X 0,Y 425.271,Z 262.323,A -85,B 0,C 180,E1 -9758.902,E2 -9758.902} C_VEL
LIN {X 0,Y 425.251,Z 262.325,A -85,B 0,C 180,E1 -9762.656,E2 -9762.656} C_VEL
LIN {X 0,Y 425.28,Z 262.324,A -85,B 0,C 180,E1 -9765.284,E2 -9765.284} C_VEL
LIN {X 0,Y 425.243,Z 262.327,A -85,B 0,C 180,E1 -9768.619,E2 -9768.619} C_VEL
LIN {X 0,Y 425.271,Z 262.325,A -85,B 0,C 180,E1 -9771.099,E2 -9771.099} C_VEL
LIN {X 0,Y 425.286,Z 262.323,A -85,B 0,C 180,E1 -9774.664,E2 -9774.664} C_VEL
LIN {X 0,Y 425.242,Z 262.325,A -85,B 0,C 180,E1 -9778.072,E2 -9778.072} C_VEL
LIN {X 0,Y 425.288,Z 262.322,A -85,B 0,C 180,E1 -9781.365,E2 -9781.365} C_VEL
LIN {X 0,Y 425.313,Z 262.359,A -85,B 0,C 180,E1 -9784.228,E2 -9784.228} C_VEL
LIN {X 0,Y 427.108,Z 272.528,A -85,B 0,C 180,E1 -9786.483,E2 -9786.483} C_VEL
LIN {X 0,Y 426.43,Z 287.073,A -85,B 0,C 180,E1 -9789.5,E2 -9789.5} C_VEL
LIN {X 0,Y 425.722,Z 302.756,A -85,B 0,C 180,E1 -9792.714,E2 -9792.714} C_VEL
LIN {X 0,Y 425.235,Z 315.466,A -85,B 0,C 180,E1 -9795.261,E2 -9795.261} C_VEL
LIN {X 0,Y 427.927,Z 338.194,A -85,B 0,C 180,E1 -9795.739,E2 -9795.739} C_VEL
LIN {X 0,Y 427.554,Z 392.316,A -85,B 0,C 180,E1 -9796.664,E2 -9796.664} C_VEL
LIN {X 0,Y 427.295,Z 401.607,A -85,B 0,C 180,E1 -9796.93,E2 -9796.93} C_VEL
LIN {X 0,Y 426.953,Z 410.072,A -85,B 0,C 180,E1 -9797.282,E2 -9797.282} C_VEL
LIN {X 0,Y 426.586,Z 418.587,A -85,B 0,C 180,E1 -9797.754,E2 -9797.754} C_VEL
LIN {X 0,Y 426.157,Z 426.94,A -85,B 0,C 180,E1 -9798.345,E2 -9798.345} C_VEL
LIN {X 0,Y 425.738,Z 435.008,A -85,B 0,C 180,E1 -9799.057,E2 -9799.057} C_VEL
LIN {X 0,Y 425.29,Z 443.724,A -85,B 0,C 180,E1 -9800.008,E2 -9800.008} C_VEL
LIN {X 0,Y 424.81,Z 452.281,A -85,B 0,C 180,E1 -9801.198,E2 -9801.198} C_VEL
LIN {X 0,Y 424.561,Z 459.007,A -85,B 0,C 180,E1 -9802.391,E2 -9802.391} C_VEL
LIN {X 0,Y 424.388,Z 463.424,A -85,B 0,C 180,E1 -9803.344,E2 -9803.344} C_VEL
LIN {X 0,Y 424.236,Z 467.101,A -85,B 0,C 180,E1 -9804.296,E2 -9804.296} C_VEL
LIN {X 0,Y 424.235,Z 470.124,A -85,B 0,C 180,E1 -9805.249,E2 -9805.249} C_VEL
LIN {X 0,Y 424.158,Z 472.465,A -85,B 0,C 180,E1 -9806.2,E2 -9806.2} C_VEL
LIN {X 0,Y 424.236,Z 474.233,A -85,B 0,C 180,E1 -9807.152,E2 -9807.152} C_VEL
LIN {X 0,Y 424.188,Z 475.493,A -85,B 0,C 180,E1 -9808.102,E2 -9808.102} C_VEL
LIN {X 0,Y 424.176,Z 476.278,A -85,B 0,C 180,E1 -9809.051,E2 -9809.051} C_VEL
LIN {X 0,Y 424.197,Z 476.576,A -85,B 0,C 180,E1 -9810,E2 -9810} C_VEL
LIN {X 0,Y 424.177,Z 476.276,A -85,B 0,C 180,E1 -9810.95,E2 -9810.95} C_VEL
LIN {X 0,Y 424.188,Z 475.487,A -85,B 0,C 180,E1 -9811.899,E2 -9811.899} C_VEL
LIN {X 0,Y 424.236,Z 474.223,A -85,B 0,C 180,E1 -9812.849,E2 -9812.849} C_VEL
LIN {X 0,Y 424.175,Z 471.287,A -85,B 0,C 180,E1 -9814.276,E2 -9814.276} C_VEL
LIN {X 0,Y 424.257,Z 468.619,A -85,B 0,C 180,E1 -9815.228,E2 -9815.228} C_VEL
LIN {X 0,Y 424.329,Z 464.415,A -85,B 0,C 180,E1 -9816.406,E2 -9816.406} C_VEL
LIN {X 0,Y 424.558,Z 458.973,A -85,B 0,C 180,E1 -9817.61,E2 -9817.61} C_VEL
LIN {X 0,Y 424.81,Z 452.245,A -85,B 0,C 180,E1 -9818.803,E2 -9818.803} C_VEL
LIN {X 0,Y 425.291,Z 443.68,A -85,B 0,C 180,E1 -9819.993,E2 -9819.993} C_VEL
LIN {X 0,Y 425.739,Z 434.95,A -85,B 0,C 180,E1 -9820.944,E2 -9820.944} C_VEL
LIN {X 0,Y 426.146,Z 426.863,A -85,B 0,C 180,E1 -9821.656,E2 -9821.656} C_VEL
LIN {X 0,Y 426.608,Z 418.493,A -85,B 0,C 180,E1 -9822.246,E2 -9822.246} C_VEL
LIN {X 0,Y 426.933,Z 409.947,A -85,B 0,C 180,E1 -9822.72,E2 -9822.72} C_VEL
LIN {X 0,Y 427.307,Z 400.6,A -85,B 0,C 180,E1 -9823.101,E2 -9823.101} C_VEL
LIN {X 0,Y 427.65,Z 389.373,A -85,B 0,C 180,E1 -9823.396,E2 -9823.396} C_VEL
LIN {X 0,Y 427.843,Z 337.8,A -85,B 0,C 180,E1 -9824.265,E2 -9824.265} C_VEL
LIN {X 0,Y 425.221,Z 315.186,A -85,B 0,C 180,E1 -9824.752,E2 -9824.752} C_VEL
LIN {X 0,Y 425.984,Z 296.695,A -85,B 0,C 180,E1 -9828.518,E2 -9828.518} C_VEL
LIN {X 0,Y 426.811,Z 279.774,A -85,B 0,C 180,E1 -9832.001,E2 -9832.001} C_VEL
LIN {X 0,Y 427.083,Z 272.487,A -85,B 0,C 180,E1 -9833.519,E2 -9833.519} C_VEL
LIN {X 0,Y 425.303,Z 262.323,A -85,B 0,C 180,E1 -9835.773,E2 -9835.773} C_VEL
LIN {X 0,Y 425.295,Z 262.32,A -85,B 0,C 180,E1 -9838.858,E2 -9838.858} C_VEL
LIN {X 0,Y 425.245,Z 262.324,A -85,B 0,C 180,E1 -9841.929,E2 -9841.929} C_VEL
LIN {X 0,Y 425.289,Z 262.323,A -85,B 0,C 180,E1 -9845.337,E2 -9845.337} C_VEL
LIN {X 0,Y 425.264,Z 262.326,A -85,B 0,C 180,E1 -9848.903,E2 -9848.903} C_VEL
LIN {X 0,Y 425.262,Z 262.322,A -85,B 0,C 180,E1 -9851.954,E2 -9851.954} C_VEL
LIN {X 0,Y 425.285,Z 262.321,A -85,B 0,C 180,E1 -9855.283,E2 -9855.283} C_VEL
